// TwinCAT 3 PLC project FMS_205
// ProgramVersion: 3.1.4023.0
// libraries:
//   Tc2_Standard, * (Beckhoff Automation GmbH)
//   Tc2_System, * (Beckhoff Automation GmbH)
//   Tc3_Module, * (Beckhoff Automation GmbH)
//   VisuDialogs, * (System)
// project tree:
//   DUTs/ CaracteristicasPieza.TcDUT, E_GEMMA.TcTLEO, Pieza.TcDUT
//   / GlobalTextList.TcGTLO, PlcTask.TcTTO, Visualization Manager.TcVMO (not stored)
//   GVLs/ Constantes.TcGVL
//   POUs/Estacion/ FB_Coordinador_SFC.TcPOU, FB_Director.TcPOU, FB_Estacion.TcPOU
//   POUs/FBs/ FB_Clock.TcPOU
//   POUs/Funciones/ AjustarIndice.TcPOU
//   POUs/ MAIN.TcPOU
//   POUs/Tareas/ FB_AvanzarAlimentador_SFC.TcPOU, FB_EstacionVaciar_SFC.TcPOU, FB_EstacionRestaurar_SFC.TcPOU, FB_Medir_SFC.TcPOU, FB_EmpujarPlato_SFC.TcPOU, FB_RechazarPieza_SFC.TcPOU, FB_DescargarPieza_SFC.TcPOU, FB_SituarPale_SFC.TcPOU, FB_CargarPieza_SFC.TcPOU, FB_TransferirPale_SFC.TcPOU, FB_RetrocederPlato_SFC.TcPOU
//   VISUs/ Visualization.TcVIS
// real-time tasks:
//   TASK PlcTask: cycle T#10ms, priority 20, ADS port 350
// I/O:
//   DEVICE Device 1 (EtherCAT), AmsNetId 192.168.109.1.2.1
//     Term 1 (EK1200) [EK1200-5000 EtherCAT Power supply (2A E-Bus)]
//       Term 2 (EL1008) [EL1008 8Ch. Dig. Input 24V, 3ms]
//       Term 3 (EL1008) [EL1008 8Ch. Dig. Input 24V, 3ms]
//       Term 4 (EL2008) [EL2008 8Ch. Dig. Output 24V, 0.5A]
//       Term 5 (EL2008) [EL2008 8Ch. Dig. Output 24V, 0.5A]
//       Term 6 (EL1008) [EL1008 8Ch. Dig. Input 24V, 3ms]
//       Term 7 (EL1008) [EL1008 8Ch. Dig. Input 24V, 3ms]
//       Term 8 (EL2008) [EL2008 8Ch. Dig. Output 24V, 0.5A]
//       Term 9 (EL2008) [EL2008 8Ch. Dig. Output 24V, 0.5A]
//       Term 10 (EL5151) [EL5151 1Ch. Inc. Encoder]
//       Term 11 (EL9011) [EL9011 End Terminal]
//   DEVICE Device 3 (RT-Ethernet Protocol), AmsNetId 192.168.109.1.4.1
//   DEVICE Device 2 (NOV-DP-RAM)
// variable links:
//   FMS_205/FMS_205 Instance <-> Device 1 (EtherCAT)/Term 1 (EK1200)/Term 10 (EL5151)
//     PlcTask Inputs/MAIN.Estacion.Codificador <-> ENC Inputs/Counter value
//   FMS_205/FMS_205 Instance <-> Device 1 (EtherCAT)/Term 1 (EK1200)/Term 2 (EL1008)
//     PlcTask Inputs/MAIN.Estacion.CodigoPaleBit0 <-> Channel 7/CodigoPaleBit0
//     PlcTask Inputs/MAIN.Estacion.CodigoPaleBit1 <-> Channel 8/CodigoPaleBit1
//     PlcTask Inputs/MAIN.Estacion.EstacionConectada <-> Channel 5/EstacionConectada
//     PlcTask Inputs/MAIN.Estacion.PresenciaPale <-> Channel 6/PresenciaPale
//     PlcTask Inputs/MAIN.Estacion.PulsadorEmergencia <-> Channel 1/PulsadorEmergencia
//     PlcTask Inputs/MAIN.Estacion.PulsadorMarcha <-> Channel 3/PulsadorMarcha
//     PlcTask Inputs/MAIN.Estacion.PulsadorParada <-> Channel 4/PulsadorParada
//     PlcTask Inputs/MAIN.Estacion.SelectorManual <-> Channel 2/SelectorManual
//   FMS_205/FMS_205 Instance <-> Device 1 (EtherCAT)/Term 1 (EK1200)/Term 3 (EL1008)
//     PlcTask Inputs/MAIN.Estacion.CodigoPaleBit2 <-> Channel 1/CodigoPaleBit2
//   FMS_205/FMS_205 Instance <-> Device 1 (EtherCAT)/Term 1 (EK1200)/Term 4 (EL2008)
//     PlcTask Outputs/MAIN.Estacion.CintaActiva <-> Channel 5/CintaActiva
//     PlcTask Outputs/MAIN.Estacion.CintaInvierte <-> Channel 6/CintaInvierte
//     PlcTask Outputs/MAIN.Estacion.DesconectaEstacion <-> Channel 1/DesconectaEstacion
//     PlcTask Outputs/MAIN.Estacion.LamparaAlarma <-> Channel 2/LamparaAlarma
//     PlcTask Outputs/MAIN.Estacion.LamparaMarcha <-> Channel 3/LamparaMarcha
//     PlcTask Outputs/MAIN.Estacion.LamparaMaterial <-> Channel 4/LamparaMaterial
//     PlcTask Outputs/MAIN.Estacion.RetenedorBaja <-> Channel 7/RetenedorBaja
//     PlcTask Outputs/MAIN.Estacion.SeparadorSube <-> Channel 8/Output
//   FMS_205/FMS_205 Instance <-> Device 1 (EtherCAT)/Term 1 (EK1200)/Term 5 (EL2008)
//     PlcTask Outputs/MAIN.Estacion.AvisadorSonoro <-> Channel 1/AvisadorSonoro
//   FMS_205/FMS_205 Instance <-> Device 1 (EtherCAT)/Term 1 (EK1200)/Term 6 (EL1008)
//     PlcTask Inputs/MAIN.Estacion.CargadorAbajo <-> Channel 4/CargadorAbajo
//     PlcTask Inputs/MAIN.Estacion.CargadorArriba <-> Channel 3/CargadorArriba
//     PlcTask Inputs/MAIN.Estacion.CargadorDelante <-> Channel 2/CargadorDelante
//     PlcTask Inputs/MAIN.Estacion.CargadorDetras <-> Channel 1/CargadorDetras
//     PlcTask Inputs/MAIN.Estacion.PlatoEmpujadorDetras <-> Channel 5/PlatoEmpujadorDetras
//     PlcTask Inputs/MAIN.Estacion.RechazadorArriba <-> Channel 8/RechazadorArriba
//     PlcTask Inputs/MAIN.Estacion.RechazadorDelante <-> Channel 7/RechazadorDelante
//     PlcTask Inputs/MAIN.Estacion.RechazadorDetras <-> Channel 6/RechazadorDetras
//   FMS_205/FMS_205 Instance <-> Device 1 (EtherCAT)/Term 1 (EK1200)/Term 7 (EL1008)
//     PlcTask Inputs/MAIN.Estacion.AlimentadorDelante <-> Channel 6/AlimentadorDelante
//     PlcTask Inputs/MAIN.Estacion.DescargadorAbajo <-> Channel 5/DescargadorAbajo
//     PlcTask Inputs/MAIN.Estacion.DescargadorArriba <-> Channel 4/DescargadorArriba
//     PlcTask Inputs/MAIN.Estacion.DescargadorDelante <-> Channel 3/DescaradorDelante
//     PlcTask Inputs/MAIN.Estacion.DescargadorDetras <-> Channel 2/DescargadorDetras
//     PlcTask Inputs/MAIN.Estacion.DetectorFotoelectrico <-> Channel 8/DetectorFotoelectrico
//     PlcTask Inputs/MAIN.Estacion.DetectorInductivo <-> Channel 7/DetectorInductivo
//     PlcTask Inputs/MAIN.Estacion.RechazadorVacio <-> Channel 1/RechazadorVacio
//   FMS_205/FMS_205 Instance <-> Device 1 (EtherCAT)/Term 1 (EK1200)/Term 8 (EL2008)
//     PlcTask Outputs/MAIN.Estacion.CargadorAvanza <-> Channel 1/CargadorAvanza
//     PlcTask Outputs/MAIN.Estacion.CargadorBaja <-> Channel 2/CargadorBaja
//     PlcTask Outputs/MAIN.Estacion.CargadorCierra <-> Channel 3/CargadorCierra
//     PlcTask Outputs/MAIN.Estacion.PlatoEmpujadorAvanza <-> Channel 4/PlatoEmpujadorAvanza
//     PlcTask Outputs/MAIN.Estacion.PlatoRetenedorAtras <-> Channel 5/PlatoRetenedorAtras
//     PlcTask Outputs/MAIN.Estacion.RechazadorAvanza <-> Channel 6/RechazadorAvanza
//     PlcTask Outputs/MAIN.Estacion.RechazadorBaja <-> Channel 8/RechazadorBaja
//     PlcTask Outputs/MAIN.Estacion.RechazadorRetrocede <-> Channel 7/RechazadorRetrocede
//   FMS_205/FMS_205 Instance <-> Device 1 (EtherCAT)/Term 1 (EK1200)/Term 9 (EL2008)
//     PlcTask Outputs/MAIN.Estacion.AlimentadorAvanza <-> Channel 5/AlimentadorAvanza
//     PlcTask Outputs/MAIN.Estacion.DescargadorAvanza <-> Channel 2/DescargadorAvanza
//     PlcTask Outputs/MAIN.Estacion.DescargadorBaja <-> Channel 3/DescargadorBaja
//     PlcTask Outputs/MAIN.Estacion.DescargadorCierra <-> Channel 4/DescargadorCierra
//     PlcTask Outputs/MAIN.Estacion.MedidorBaja <-> Channel 6/MedidorBaja
//     PlcTask Outputs/MAIN.Estacion.RechazadorSucciona <-> Channel 1/RechazadorSucciona

CONFIGURATION FMS_205
    RESOURCE PLC ON TwinCAT3
        TASK PlcTask(INTERVAL := T#10ms, PRIORITY := 20);
        PROGRAM MAIN WITH PlcTask : MAIN;
    END_RESOURCE
END_CONFIGURATION

// ---- DUTs/CaracteristicasPieza.TcDUT
TYPE CaracteristicasPieza:
STRUCT
    Claro     : BOOL := FALSE;
    Metalico  : BOOL := FALSE;
	Alta : BOOL := FALSE;				//1290 Alta , 1370 baja. Reves: >1685 No hay >2000
END_STRUCT
END_TYPE

// ---- DUTs/E_GEMMA.TcTLEO
{attribute 'qualified_only'}
{attribute 'strict'}
TYPE E_GEMMA :
(
    // Modos de la Guia de Estudio de los Modos de Marcha y Parada
    // Modes du Guide d'Etude des Modes de Marche et d'Arrêt
    // Modes of Study Guide of the Modes of Operating and Stopping

    // Procedimientos de parada [Les procédures d'arrets - Stop procedure
    A1, //  0: Parada en el estado inicial 
        //  0: Arrêt dans etat initial
        //  0: Stopped in the initial state
    A2, //  1: Parada solicitada a final de ciclo 
        //  1: Arret demandé en fin de cycle
        //  1: Requested end cycle stop
    A3, //  2: Parada solicitada en un estado determinado 
        //  2: Arret demande dans etat determine
        //  2: Requested particular state stop
    A4, //  3: Parada obtenida 
        //  3: Arret obtenu 
        //  3: Obteined stop
    A5, //  4: Preparacion para la recuperacion del fallo 
        //  4: Preparation pour remise en route apres defaillance
        //  4: Preparation for the recovery of the failure
    A6, //  5: Situando la PO en el estado inicial 
        //  5: Mise PO dans état initial 
        //  5: Set the PO in initial state
    A7, //  6: Situando la PO en un estado determinado 
        //  6: Mise PO dans état déterminé 
        //  6: Set the PO in a certain state

    // Procedimientos de funcionamiento 
    // Les procédures de fonctionnement 
    // Operating procedures
    F1, //  7: Produccion normal 
        //  7: Production normale 
        //  7: Normal operation
    F2, //  8: Secuencia de preparacion 
        //  8: Marche de preparation 
        //  8: Preparation sequence
    F3, //  9: Secuencia de finalizacion 
        //  9: Marche de cloture
        //  9: Ending sequence
    F4, // 10: Verificacion en desorden 
        // 10: Marche de verification dans le desordre 
        // 10: Verification with no order
    F5, // 11: Verificacion en orden 
        // 11: Marche de verification dans l'ordre 
        // 11: Verification whit order
    F6, // 12: Secuencia de prueba 
        // 12: Marche de test 
        // 12:Test sequence

    // Procedimientos de fallo 
    // es procédures en défaillances
    // Failure procedures
    D1, // 13: Parada de emergencia 
        // 13: Arret d'urgence 
        // 13: Emergency stop
    D2, // 14: Diagnostico y/o tratamiento de los fallos 
        // 14: Diagnostic et/ou traitement de la défaillance 
        // 14: Diagnosis and/or treatment of failures
    D3  // 15: Produccion a pesar de los fallos 
        // 15: Production tout de même 
        // 15: Production despite the failures
);
END_TYPE

// ---- DUTs/Pieza.TcDUT
TYPE Pieza:
STRUCT
    TipoPieza : CaracteristicasPieza;		
	BienColocada    : BOOL := FALSE;
	EsBuena : BOOL := FALSE;
END_STRUCT
END_TYPE

// ---- GVLs/Constantes.TcGVL
VAR_GLOBAL CONSTANT
	TAMANO_LISTA_PIEZAS : UINT := 8;
	TAMANO_LISTA_CONDICIONES : UINT := 6;
END_VAR

// ---- POUs/MAIN.TcPOU
PROGRAM MAIN
//Ingenieria Electronica Robotica y Mecatronica (GIERM)
//Autmatizacion Industrial
//FMS205 
//GEMMA
//Grupo 03
//Paula Chova Garcia
//Jose Luis Perez Martin
//Tobias Garibaldi Thwaites Rayner


VAR
    Estacion: FB_Estacion;
END_VAR

Estacion();

END_PROGRAM

// ---- POUs/Estacion/FB_Estacion.TcPOU
FUNCTION_BLOCK FB_Estacion
// FMS-203 - Estructurado
VAR CONSTANT
	
END_VAR
VAR_INPUT
    // Parametros de control de la estacion
    CicloACiclo: BOOL := 0;
	PausaEstado: BOOL;
    ReiniciaEstado: BOOL;   
	FinCiclo: BOOL := FALSE;
	PiezaAPieza: BOOL := FALSE;
	FinPieza: BOOL:= FALSE;
	Fallo: BOOL := FALSE;
	FaltaMaterial : BOOL := FALSE;

    // Parametros de control de la tarea
    UnidadesSolicitadas: UINT := 1;
    
	//Variables auxiliares
	NCiclos : INT := 0;
	
    // Parametros de tiempo
    TpoPinza: TIME := T#1S;
	TpoRechazador: TIME := T#1S;
	TpoEmpujadorAvanza: TIME := T#1S;
    TpoPaleEntrada: TIME := T#1S;
	TpoPaleSalida : TIME := T#1S;
	TpoCintaRetenedor : TIME := T#1S;
	TpoPaleTransferencia : TIME := T#1S;
	TpoAlimentador: TIME := T#1300MS;
    TpoMedidor: TIME := T#1S;
	TpoPreparacion: TIME := T#1S;
	TpoFinalizacion : TIME := T#2S;
    
END_VAR

VAR_OUTPUT
	  // Parametros de; estado de la estacion
    CondicionInicial: BOOL;
    CondicionMarcha: BOOL;
	PrepararProduccion: BOOL := FALSE;
	FinalizarProduccion: BOOL := FALSE;
    CodigoPale: BYTE;  
    
    // Parametros de control de la tarea 
    UnidadesPendientes: UINT := 0;
    UnidadesRealizadas: UINT :=0;
	
	 // Entradas comunes
    PulsadorEmergencia AT %I*: BOOL;
    SelectorManual AT %I*: BOOL;
    PulsadorMarcha AT %I*: BOOL;
    PulsadorParada AT %I*: BOOL := TRUE; // Contacto normalmente cerrado
    EstacionConectada AT %I*: BOOL := TRUE;
    PresenciaPale AT %I*: BOOL;
    CodigoPaleBit0 AT %I*: BOOL;
    CodigoPaleBit1 AT %I*: BOOL;
    CodigoPaleBit2 AT %I*: BOOL;

    // Entradas espeficicas
    CargadorDetras AT %I*: BOOL;
	CargadorDelante AT %I*: BOOL;
	CargadorArriba AT %I*: BOOL;
	CargadorAbajo AT %I*: BOOL;
	PlatoEmpujadorDetras AT %I*: BOOL;
	RechazadorDetras AT %I*: BOOL;
	RechazadorDelante AT %I*: BOOL;
	RechazadorArriba AT %I*: BOOL;
	
	RechazadorVacio AT %I*: BOOL;
	DescargadorDetras AT %I*: BOOL;
	DescargadorDelante AT %I*: BOOL;
	DescargadorArriba AT %I*: BOOL;
	DescargadorAbajo AT %I*: BOOL;
	AlimentadorDelante AT %I*: BOOL := FALSE;
	DetectorInductivo AT %I*: BOOL;
	DetectorFotoelectrico AT %I*: BOOL;
	Codificador AT %I*: UINT;
END_VAR

VAR
	ModoAnterior: E_GEMMA; 
	
	 // Bloques funcionales
	CLK: FB_Clock;
	
	Director: FB_Director;
    Coordinador: FB_Coordinador_SFC;
	
	Restaurar: FB_EstacionRestaurar_SFC;
    Vaciar: FB_EstacionVaciar_SFC;
	AvanzarAlimentador: FB_AvanzarAlimentador_SFC;
    SituarPale: FB_SituarPale_SFC;
    CargarPieza: FB_CargarPieza_SFC;
	EmpujarPlato: FB_EmpujarPlato_SFC;
	RetrocederPlato : FB_RetrocederPlato_SFC;
    DescargarPieza: FB_DescargarPieza_SFC;
    RechazarPieza: FB_RechazarPieza_SFC;
    TransferirPale: FB_TransferirPale_SFC;
	Medir: FB_Medir_SFC;
	
	// Arrays
	ListadePiezas: ARRAY[1..TAMANO_LISTA_PIEZAS] OF Pieza; // Array de tamaño 8 piezas 
	ListaPiezasSolicitadas: ARRAY[1..TAMANO_LISTA_CONDICIONES] OF UINT
 	:= [TAMANO_LISTA_CONDICIONES(0)]; 
	
    // Salidas comunes
    DesconectaEstacion AT %Q*: BOOL;
    LamparaAlarma AT %Q*: BOOL;
    LamparaMarcha AT %Q*: BOOL;
	LamparaMaterial AT %Q*: BOOL;
    CintaActiva AT %Q*: BOOL;
    CintaInvierte AT %Q*: BOOL;
    RetenedorBaja AT %Q*: BOOL;
	
	AvisadorSonoro AT %Q*: BOOL;

    // Salidas especificas
    CargadorAvanza AT %Q*: BOOL;
	CargadorBaja AT %Q*: BOOL; 	
	CargadorCierra AT %Q*: BOOL;
	PlatoEmpujadorAvanza AT %Q*: BOOL;
	PlatoRetenedorAtras AT %Q*: BOOL;
	RechazadorAvanza AT %Q*: BOOL;
	RechazadorRetrocede AT %Q*: BOOL;
	RechazadorBaja AT %Q*: BOOL;
	
	RechazadorSucciona AT %Q*: BOOL;
	DescargadorAvanza AT %Q*: BOOL;
	DescargadorBaja AT %Q*: BOOL;
	DescargadorCierra AT %Q*: BOOL;
	AlimentadorAvanza AT %Q*: BOOL;
	MedidorBaja AT %Q*: BOOL;
	SeparadorSube AT %Q*: BOOL;	
	
	PlatoEmpujado: BOOL;
	PiezaRechazada: BOOL;
END_VAR

Director(
	CondicionInicial := CondicionInicial,
    CondicionMarcha := CondicionMarcha,
	Emergencia := PulsadorEmergencia,
    FaltaPreparacion := (UnidadesRealizadas = 0) AND Director.Modo = E_GEMMA.A1,
    FinTarea := (UnidadesPendientes = 0),
    FinCiclo := Coordinador.Done,
	FinPieza := FinPieza,
    Manual := SelectorManual,
    Marcha := PulsadorMarcha,
    ParaCiclo := NOT PulsadorParada,
    Preparada := Vaciar.Done,
    Reinicia := ReiniciaEstado,
	PrepararProduccion := PrepararProduccion,
    FinalizarProduccion := FinalizarProduccion,
	Fallo := Fallo
);

// MODO AUTOMATICO
IF (Director.Modo <> E_GEMMA.F4) THEN
    // Bloques funcionales
    Coordinador(
        SFCPause := NOT ReiniciaEstado AND PausaEstado, 
        // OR Director.Modo := E_GEMMA.F3 
        SFCReset := ReiniciaEstado,
        Ack := TRUE,
        Execute :=  (Director.Modo = E_GEMMA.F1),
        Resume := PulsadorMarcha,
        StepByStep := CicloaCiclo,
		FinCiclo := FinCiclo,
		FinPieza => FinPieza,
		PiezaAPieza := PiezaAPieza,
        PaleSituado := SituarPale.Done,
		AlimentadorAvanzado := AvanzarAlimentador.Done,
        PiezaCargada := CargarPieza.Done,
        PlatoEmpujado := EmpujarPlato.Done,
		PlatoRetrocedido := RetrocederPlato.Done,
        PiezaDescargada := DescargarPieza.Done,
        PiezaRechazada := RechazarPieza.Done,
		PiezaMedida := Medir.Done,
        PaleTransferido := TransferirPale.Done,
        CondicionInicial := CondicionInicial,
        UnidadesSolicitadas => UnidadesSolicitadas,
		UnidadesRealizadas => UnidadesRealizadas,
		UnidadesPendientes => UnidadesPendientes,
		ListadePiezas := ListadePiezas,
		ListaPiezasSolicitadas := ListaPiezasSolicitadas,
		Fallo => Fallo,
		FaltaMaterial := FaltaMaterial
        );
        
    SituarPale(
        SFCPause := NOT ReiniciaEstado AND PausaEstado,
        SFCReset := ReiniciaEstado,
        Ack := NOT Coordinador.SituaPale,
        Execute := Coordinador.SituaPale,
        TpoPaleEntrada := TpoPaleEntrada,
        PresenciaPale := PresenciaPale,
        CodigoPaleBit0 := CodigoPaleBit0,
        CodigoPaleBit1 := CodigoPaleBit1,
        CodigoPaleBit2 := CodigoPaleBit2
        );
        
	 AvanzarAlimentador(
        SFCPause := NOT ReiniciaEstado AND PausaEstado,
        SFCReset := ReiniciaEstado,
        Ack := NOT Coordinador.AvanzaAlimentador,
        Execute := Coordinador.AvanzaAlimentador,
		TpoAlimentador :=  TpoAlimentador,
        AlimentadorDelante := AlimentadorDelante,
		PulsadorMarcha := PulsadorMarcha,
		Fallo => Fallo,
		FaltaMaterial := FaltaMaterial
        );	
	

    CargarPieza(
        SFCPause := NOT ReiniciaEstado AND PausaEstado,
        SFCReset := ReiniciaEstado,
        Ack := NOT Coordinador.CargaPieza,
        Execute := Coordinador.CargaPieza,
		TpoPinza :=  TpoPinza,
        CargadorDetras := CargadorDetras,
		CargadorDelante := CargadorDelante,
		CargadorArriba := CargadorArriba,
		CargadorAbajo := CargadorAbajo
        );
        
     EmpujarPlato(
        SFCPause := NOT ReiniciaEstado AND PausaEstado,
        SFCReset := ReiniciaEstado,
        Ack := NOT Coordinador.EmpujaPlato AND NOT Vaciar.EmpujaPlato,
        Execute := Coordinador.EmpujaPlato OR Vaciar.EmpujaPlato,
		TpoEmpujadorAvanza := TpoEmpujadorAvanza,
        );
	
	RetrocederPlato(
        SFCPause := NOT ReiniciaEstado AND PausaEstado,
        SFCReset := ReiniciaEstado,
        Ack := NOT Coordinador.RetrocederPlato,
        Execute := Coordinador.RetrocederPlato,
		TpoEmpujadorAvanza :=  TpoEmpujadorAvanza,
        PlatoEmpujadorDetras := PlatoEmpujadorDetras,
        );
		
    
    DescargarPieza(
        SFCPause := NOT ReiniciaEstado AND PausaEstado,
        SFCReset := ReiniciaEstado,
        Ack := NOT Coordinador.DescargaPieza,
        Execute := Coordinador.DescargaPieza,
        TpoPinza :=  TpoPinza,
        DescargadorDetras := DescargadorDetras,
        DescargadorDelante := DescargadorDelante,
        DescargadorArriba := DescargadorArriba,
        DescargadorAbajo := DescargadorAbajo
        );
    
    RechazarPieza(
        SFCPause := NOT ReiniciaEstado AND PausaEstado,
        SFCReset := ReiniciaEstado,
        Ack := NOT Coordinador.RechazaPieza AND NOT Vaciar.RechazaPieza,
        Execute := Coordinador.RechazaPieza OR Vaciar.RechazaPieza,
		TpoRechazador := TpoRechazador,
        RechazadorDetras := RechazadorDetras,
        RechazadorDelante := RechazadorDelante,
        RechazadorArriba := RechazadorArriba,
		RechazadorVacio := RechazadorVacio,
		PulsadorMarcha := PulsadorMarcha,
		Fallo => Fallo
        );
		
	 Medir(
        SFCPause := NOT ReiniciaEstado AND PausaEstado,
        SFCReset := ReiniciaEstado,
        Ack := NOT Coordinador.MedidorMide,
        Execute := Coordinador.MedidorMide,
		TpoMedidor := TpoMedidor,
        Codificador := Codificador,
        DetectorFotoelectrico := DetectorFotoelectrico,
        DetectorInductivo := DetectorInductivo,
		NCiclos := NCiclos,
		ListadePiezas := ListadePiezas,
        );
    
    TransferirPale(
        SFCPause := NOT ReiniciaEstado AND PausaEstado,
        SFCReset := ReiniciaEstado,
        Ack := NOT Coordinador.TransfierePale,
        Execute := Coordinador.TransfierePale,
        TpoCintaRetenedor := TpoCintaRetenedor,
        TpoPaleSalida := TpoPaleSalida,
        TpoPaleTransferencia := TpoPaleTransferencia,
        PresenciaPale := PresenciaPale
        );
    Restaurar(
        SFCPause := NOT ReiniciaEstado AND PausaEstado,
        SFCReset := ReiniciaEstado,
        Ack := TRUE,
        Execute := (Director.Modo = E_GEMMA.A6),
        CargadorDetras := CargadorDetras,
        PlatoEmpujadorDetras := PlatoEmpujadorDetras,
        DescargadorDetras := DescargadorDetras,
		RechazadorDetras := RechazadorDetras
        );
	Vaciar(
        SFCPause := NOT ReiniciaEstado AND PausaEstado,
        SFCReset := ReiniciaEstado,
        Ack := (Director.Modo <> E_GEMMA.F2) AND (Director.Modo <> E_GEMMA.F3),
        Execute := (Director.Modo = E_GEMMA.F2) OR (Director.Modo = E_GEMMA.F3),
		TpoPreparacion := TpoPreparacion,
        TpoMedidor := TpoMedidor,
		PlatoEmpujado := EmpujarPlato.Done,
		PiezaRechazada := RechazarPieza.Done,
		PulsadorMarcha := PulsadorMarcha,
		Codificador := Codificador
        );
		
    // Acciones
   AvisadorSonoro := ((Director.Modo = E_GEMMA.F2) AND CLK.Q) 
        OR (Director.Modo = E_GEMMA.F3)
		OR (Director.Modo = E_GEMMA.D1)
		OR (Director.Modo = E_GEMMA.D2);   
    LamparaAlarma := (Director.Modo = E_GEMMA.D1) 
        OR ((Director.Modo = E_GEMMA.A6) AND CLK.Q)
		OR (Director.Modo = E_GEMMA.D2);
    LamparaMarcha := (Director.Produccion AND NOT Coordinador.Done)
        OR ((Director.Modo = E_GEMMA.A1) AND CLK.Q);
    

    CintaActiva := NOT PausaEstado 
        AND (SituarPale.CintaActiva OR TransferirPale.CintaActiva);
    RetenedorBaja := TransferirPale.RetenedorBaja;
	SeparadorSube := TransferirPale.SeparadorSube;
	AlimentadorAvanza := AvanzarAlimentador.AlimentadorAvanza;
    CargadorAvanza := CargarPieza.CargadorAvanza; 
    CargadorBaja := CargarPieza.CargadorBaja;    
	CargadorCierra := CargarPieza.CargadorCierra;
	PlatoEmpujadorAvanza := EmpujarPlato.PlatoEmpujadorAvanza;
	PlatoRetenedorAtras := EmpujarPlato.PlatoRetenedorAtras;
	DescargadorAvanza := DescargarPieza.DescargadorAvanza; 
    DescargadorBaja := DescargarPieza.DescargadorBaja;    
	DescargadorCierra := DescargarPieza.DescargadorCierra;
    RechazadorAvanza := RechazarPieza.RechazadorAvanza;
	RechazadorSucciona := RechazarPieza.RechazadorSucciona;
    RechazadorRetrocede := RechazarPieza.RechazadorRetrocede
	OR Restaurar.RechazadorRetrocede;
    RechazadorBaja := RechazarPieza.RechazadorBaja;
	AlimentadorAvanza := AvanzarAlimentador.AlimentadorAvanza;
	MedidorBaja := Medir.MedidorBaja OR Vaciar.MedidorBaja;
	
   
END_IF

// Parametros de salida
CondicionInicial := EstacionConectada 
    AND CargadorDetras 
    AND PlatoEmpujadorDetras
    AND DescargadorDetras
    AND RechazadorDetras;

CondicionMarcha := (UnidadesSolicitadas > 0);
NCiclos := Coordinador.NCiclos;


IF (Director.Modo <> E_GEMMA.F4) THEN
    CodigoPale := SituarPale.CodigoPale;
ELSE 
    CodigoPale.0 := CodigoPaleBit0;
    CodigoPale.1 := CodigoPaleBit1;
    CodigoPale.2 := CodigoPaleBit2;
END_IF

// ACTULIZACION DE IMAGENES
ModoAnterior := Director.Modo;

END_FUNCTION_BLOCK

// ---- POUs/FBs/FB_Clock.TcPOU
FUNCTION_BLOCK FB_Clock
(*
Square wave oscillator

Copyright (c) 2009-2017 victortorreslopez

GNU General Public License

Version history
2.1, 2017/03/15, VTL: style review (PLCopen Coding Guidelines)
2.0, 2014/12/29, VTL: complete review
1.0, 2009/11/06, VTL: first release
0.0, 2009/11/06, VTL: alfa release
*)
VAR_INPUT
  EN: BOOL := TRUE;	(* ENabled *)
  PT: TIME := T#500ms; (* Semicycle time *)
END_VAR
VAR_OUTPUT
  ET: TIME; (* Elapsed time *)
  Q: BOOL; (* Square wave *)
END_VAR
VAR
  Timer: TON; (* Auto-pilot timer *)
END_VAR

(* OUTPUT FUNCTION *)
IF Timer.Q THEN
  Q := NOT Q;
END_IF

(* FUNCTION BLOCKS *)
Timer(IN := EN AND NOT Timer.Q, PT := PT, ET => ET);

END_FUNCTION_BLOCK

// ---- POUs/Estacion/FB_Director.TcPOU
FUNCTION_BLOCK FB_Director
// FMS-203 - GEMMA

VAR_INPUT
    CondicionInicial: BOOL;
    CondicionMarcha: BOOL; 
    Emergencia: BOOL;
    FinTarea: BOOL;
    FinCiclo: BOOL;
	FinPieza: BOOL;
    Manual: BOOL;
    Marcha: BOOL;
    ParaCiclo: BOOL;
    Preparada: BOOL;
    Reinicia: BOOL;
	Fallo: BOOL;
	PrepararProduccion: BOOL;
    FinalizarProduccion: BOOL;
    FaltaPreparacion: BOOL;
END_VAR
VAR_OUTPUT
    Modo: E_GEMMA := E_GEMMA.A6;

    Defecto: BOOL; // Procedimientos de defecto
    Funcionamiento: BOOL; // Procedimientos de funcionamiento
    Parada: BOOL; // Procedimientos de parada
    Produccion: BOOL; // Procedimientos que proporcionan valor añadido
END_VAR

// FUNCION DE ESTADO
IF Emergencia THEN
    Modo := E_GEMMA.D1;
ELSIF Reinicia THEN
    Modo := E_GEMMA.A6;
ELSE
    CASE Modo OF
        // Procedimientos de parada
        E_GEMMA.A1: // Parada en el estado inicial
            IF NOT CondicionInicial THEN
                Modo := E_GEMMA.A6;
            ELSIF CondicionInicial AND CondicionMarcha AND Marcha THEN
                IF FaltaPreparacion THEN 
                    Modo := E_GEMMA.F2;
                ELSE   
                    Modo := E_GEMMA.F1;
                END_IF
            ELSIF Manual THEN
                Modo := E_GEMMA.F4;
            END_IF
        E_GEMMA.A2: // Parada solicitada a final de ciclo
           IF Marcha THEN 
               Modo := E_GEMMA.F1;
		   END_IF
        E_GEMMA.A3: // Parada solicitada en un estado determinado 
       		IF Marcha THEN 
               Modo := E_GEMMA.F1;
		   END_IF   
        E_GEMMA.A4: // Parada obtenida 
            ;
        E_GEMMA.A5: // Preparando de reanudacion tras el fallo 
            ;
        E_GEMMA.A6: // Situando el sistema en el estado inicial 
            IF CondicionInicial THEN
                Modo := E_GEMMA.A1;
            ELSIF Manual THEN
                Modo := E_GEMMA.F4;
            END_IF

        // Procedimientos de funcionamiento 
        E_GEMMA.F1: // Produccion normal 
            IF FinTarea THEN
               Modo := E_GEMMA.A6;
            ELSIF FinCiclo THEN
				Modo := E_GEMMA.F3;
			ELSIF FinPieza THEN
				Modo := E_GEMMA.A2;
			ELSIF ParaCiclo THEN
               Modo := E_GEMMA.A3;
			ELSIF Fallo THEN
				Modo := E_GEMMA.D2;
			END_IF
			
        E_GEMMA.F2: // Secuencia de preparacion 
            IF Preparada AND NOT Manual THEN
                Modo := E_GEMMA.F1;
            ELSIF Preparada AND Manual THEN
                Modo := E_GEMMA.F4;
			END_IF
        E_GEMMA.F3: // Secuencia de finalizacion 
           IF Preparada AND NOT Manual THEN
                Modo := E_GEMMA.A6;
            ELSIF Preparada AND Manual THEN
                Modo := E_GEMMA.F4;
			END_IF
        E_GEMMA.F4: // Verificacion sin orden 
            IF NOT Manual THEN
                Modo := E_GEMMA.A6;
            ELSIF (CondicionInicial) AND PrepararProduccion THEN
                Modo := E_GEMMA.F2;
            ELSIF (CondicionInicial) AND FinalizarProduccion THEN
                Modo := E_GEMMA.F3;
            END_IF
        E_GEMMA.F5: // Verificacion en orden 
            ;

        // Procedimientos de defecto 
        E_GEMMA.D1: // Parada de emergencia 
            IF NOT Emergencia THEN
                Modo := E_GEMMA.A6;
            END_IF
        E_GEMMA.D2: // Diagnostico/tratamiento de los fallos 
        IF Marcha THEN
			Modo := E_GEMMA.F1;
		END_IF    
			
    END_CASE
END_IF

// PARAMETROS DE SALIDA 
Defecto := (Modo >= E_GEMMA.D1) AND (Modo <= E_GEMMA.D3);
Funcionamiento:= (Modo >= E_GEMMA.F1);
Parada := (Modo >= E_GEMMA.A1);
Produccion := (Modo = E_GEMMA.A2) 
    OR (Modo = E_GEMMA.A3) 
    OR (Modo = E_GEMMA.F1) 
    OR (Modo = E_GEMMA.F2) 
    OR (Modo = E_GEMMA.F3) 
    OR (Modo = E_GEMMA.F5)
    OR (Modo = E_GEMMA.F6) 
    OR (Modo = E_GEMMA.D3);

END_FUNCTION_BLOCK

// ---- POUs/Estacion/FB_Coordinador_SFC.TcPOU
FUNCTION_BLOCK FB_Coordinador_SFC

VAR CONSTANT
LISTA_CONDICIONES: ARRAY[1..TAMANO_LISTA_CONDICIONES] OF CaracteristicasPieza:=[(Claro:=FALSE, Metalico:=FALSE, Alta:=TRUE), //Negra alta
					(Claro:=TRUE,Metalico:=FALSE,Alta:=TRUE), //Blanca alta					
					(Claro:=TRUE, Metalico:=TRUE, Alta:=TRUE), //Metal alta
					(Claro:=FALSE, Metalico:=FALSE, Alta:=FALSE), //Negra baja
					(Claro:=TRUE, Metalico:=FALSE, Alta:=FALSE), //Blanca baja					
					(Claro:=TRUE, Metalico:=TRUE, Alta:=FALSE)]; //Metal baja
END_VAR

VAR_IN_OUT
	ListadePiezas: ARRAY[1..TAMANO_LISTA_PIEZAS] OF Pieza; // Array de tamaño 8 piezas 
	ListaPiezasSolicitadas: ARRAY[1..TAMANO_LISTA_CONDICIONES] OF UINT; // Array de 6 condiciones (blanca, negra y metálica, de momento)
	FaltaMaterial: BOOL;
END_VAR

VAR_INPUT
	  // SFC-Flags
    SFCPause: BOOL;
    SFCReset: BOOL;
    
    // Indicadores de sincronizacion
    Ack: BOOL := TRUE;
    Execute: BOOL;
    
    // Indicadores de control
    Resume: BOOL;
    StepByStep: BOOL;
	FinCiclo: BOOL;
    PiezaAPieza: BOOL;
    // Parametros de sincronizacion
    PaleSituado: BOOL;
	AlimentadorAvanzado: BOOL;
    PiezaCargada: BOOL;
	PlatoEmpujado: BOOL;
	PiezaMedida: BOOL;
    PiezaDescargada: BOOL;
    PiezaRechazada: BOOL;
    PaleTransferido: BOOL;
	PlatoRetrocedido: BOOL;
    
    // Parametros
    CondicionInicial: BOOL;

	//Variables auxiliares
	NCiclos: INT;
	AuxNciclosDesechar: INT := 1;
	AuxNciclosDescargar: INT := 1;
	ListoParaRechazar: BOOL := FALSE;
	ListoParaDescargar: BOOL := FALSE;
	ListoParaMedir: BOOL := FALSE;
	AUX_Suma_Solicitadas: UINT;
	
END_VAR
VAR_OUTPUT
	 // Indicadores de sincronizacion
    Done: BOOL;
    Ready: BOOL;
	Fallo: BOOL;
	FinPieza: BOOL;

    // Parametros de sincronizacion
    SituaPale: BOOL;
	AvanzaAlimentador: BOOL;
	EmpujaPlato: BOOL;
	MedidorMide: BOOL;
    CargaPieza: BOOL;
    DescargaPieza: BOOL;
    RechazaPieza: BOOL;
    TransfierePale: BOOL;
	RetrocederPlato: BOOL;
    
    // Salidas
    LamparaAlarma: BOOL;
    LamparaMarcha: BOOL;
	
	//Variables
	UnidadesSolicitadas: UINT := 1;
	UnidadesPendientes: UINT;
    UnidadesRealizadas: UINT; 
	
END_VAR
VAR

END_VAR

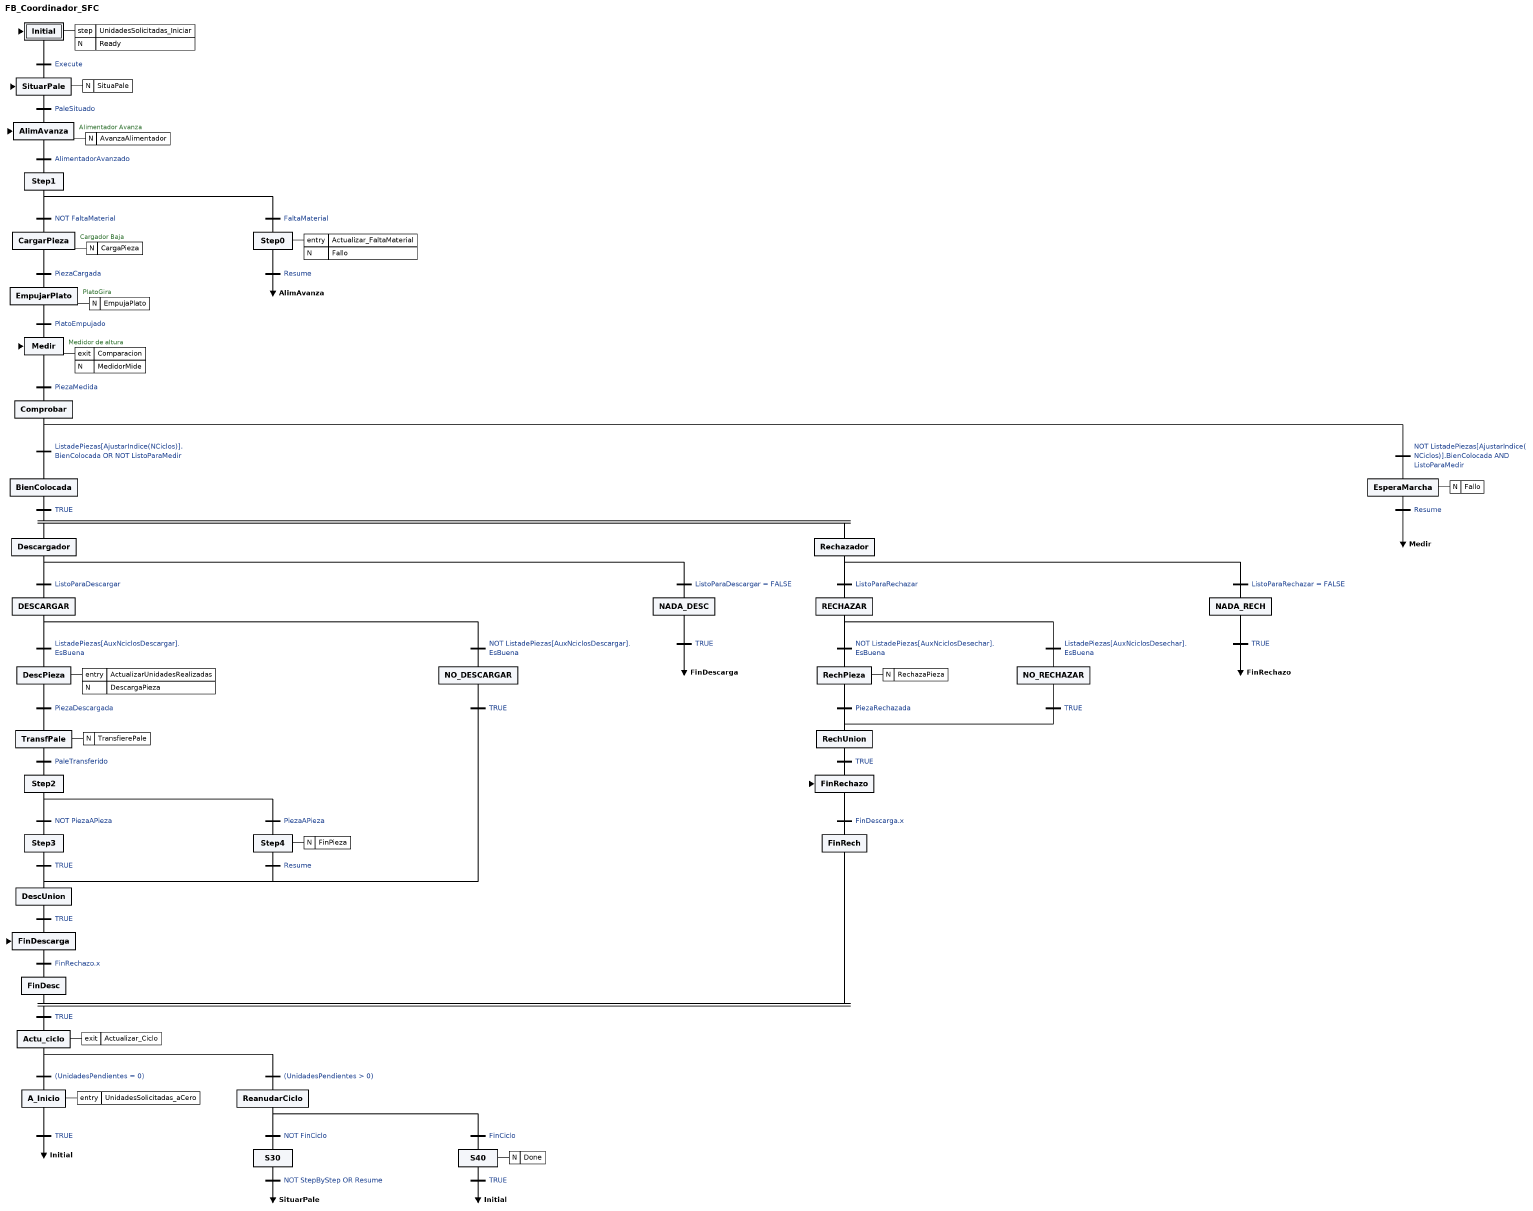
INITIAL_STEP Initial:
    UnidadesSolicitadas_Iniciar(N);  // step action
    Ready(N);
END_STEP
TRANSITION FROM Initial TO SituarPale
    := Execute;
END_TRANSITION
STEP SituarPale:
    SituaPale(N);
END_STEP
TRANSITION FROM SituarPale TO AlimAvanza
    := PaleSituado;
END_TRANSITION
// Alimentador Avanza
STEP AlimAvanza:
    AvanzaAlimentador(N);
END_STEP
TRANSITION FROM AlimAvanza TO Step1
    := AlimentadorAvanzado;
END_TRANSITION
STEP Step1:
END_STEP
TRANSITION FROM Step1 TO CargarPieza
    := NOT FaltaMaterial;
END_TRANSITION
TRANSITION FROM Step1 TO Step0
    := FaltaMaterial;
END_TRANSITION
STEP Step0:
    Actualizar_FaltaMaterial(P1);  // entry action
    Fallo(N);
END_STEP
TRANSITION FROM Step0 TO AlimAvanza
    := Resume;
END_TRANSITION
// Cargador Baja
STEP CargarPieza:
    CargaPieza(N);
END_STEP
TRANSITION FROM CargarPieza TO EmpujarPlato
    := PiezaCargada;
END_TRANSITION
// PlatoGira
STEP EmpujarPlato:
    EmpujaPlato(N);
END_STEP
TRANSITION FROM EmpujarPlato TO Medir
    := PlatoEmpujado;
END_TRANSITION
// Medidor de altura
STEP Medir:
    Comparacion(P0);  // exit action
    MedidorMide(N);
END_STEP
TRANSITION FROM Medir TO Comprobar
    := PiezaMedida;
END_TRANSITION
STEP Comprobar:
END_STEP
TRANSITION FROM Comprobar TO BienColocada
    := ListadePiezas[AjustarIndice(NCiclos)].BienColocada OR NOT ListoParaMedir;
END_TRANSITION
STEP BienColocada:
END_STEP
TRANSITION FROM BienColocada TO (Descargador, Rechazador)
    := TRUE;
END_TRANSITION
TRANSITION FROM Comprobar TO EsperaMarcha
    := NOT ListadePiezas[AjustarIndice(NCiclos)].BienColocada AND ListoParaMedir;
END_TRANSITION
STEP EsperaMarcha:
    Fallo(N);
END_STEP
TRANSITION FROM EsperaMarcha TO Medir
    := Resume;
END_TRANSITION
STEP Descargador:
END_STEP
TRANSITION FROM Descargador TO DESCARGAR
    := ListoParaDescargar;
END_TRANSITION
STEP DESCARGAR:
END_STEP
TRANSITION FROM Descargador TO NADA_DESC
    := ListoParaDescargar = FALSE;
END_TRANSITION
STEP NADA_DESC:
END_STEP
TRANSITION FROM NADA_DESC TO FinDescarga
    := TRUE;
END_TRANSITION
TRANSITION FROM DESCARGAR TO DescPieza
    := ListadePiezas[AuxNciclosDescargar].EsBuena;
END_TRANSITION
STEP DescPieza:
    ActualizarUnidadesRealizadas(P1);  // entry action
    DescargaPieza(N);
END_STEP
TRANSITION FROM DescPieza TO TransfPale
    := PiezaDescargada;
END_TRANSITION
STEP TransfPale:
    TransfierePale(N);
END_STEP
TRANSITION FROM TransfPale TO Step2
    := PaleTransferido;
END_TRANSITION
STEP Step2:
END_STEP
TRANSITION FROM Step2 TO Step3
    := NOT PiezaAPieza;
END_TRANSITION
STEP Step3:
END_STEP
TRANSITION FROM Step3 TO DescUnion
    := TRUE;
END_TRANSITION
TRANSITION FROM Step2 TO Step4
    := PiezaAPieza;
END_TRANSITION
STEP Step4:
    FinPieza(N);
END_STEP
TRANSITION FROM Step4 TO DescUnion
    := Resume;
END_TRANSITION
TRANSITION FROM DESCARGAR TO NO_DESCARGAR
    := NOT ListadePiezas[AuxNciclosDescargar].EsBuena;
END_TRANSITION
STEP NO_DESCARGAR:
END_STEP
TRANSITION FROM NO_DESCARGAR TO DescUnion
    := TRUE;
END_TRANSITION
STEP DescUnion:
END_STEP
TRANSITION FROM DescUnion TO FinDescarga
    := TRUE;
END_TRANSITION
STEP FinDescarga:
END_STEP
TRANSITION FROM FinDescarga TO FinDesc
    := FinRechazo.x;
END_TRANSITION
STEP FinDesc:
END_STEP
STEP Rechazador:
END_STEP
TRANSITION FROM Rechazador TO RECHAZAR
    := ListoParaRechazar;
END_TRANSITION
STEP RECHAZAR:
END_STEP
TRANSITION FROM Rechazador TO NADA_RECH
    := ListoParaRechazar = FALSE;
END_TRANSITION
STEP NADA_RECH:
END_STEP
TRANSITION FROM NADA_RECH TO FinRechazo
    := TRUE;
END_TRANSITION
TRANSITION FROM RECHAZAR TO RechPieza
    := NOT ListadePiezas[AuxNciclosDesechar].EsBuena;
END_TRANSITION
STEP RechPieza:
    RechazaPieza(N);
END_STEP
TRANSITION FROM RechPieza TO RechUnion
    := PiezaRechazada;
END_TRANSITION
TRANSITION FROM RECHAZAR TO NO_RECHAZAR
    := ListadePiezas[AuxNciclosDesechar].EsBuena;
END_TRANSITION
STEP NO_RECHAZAR:
END_STEP
TRANSITION FROM NO_RECHAZAR TO RechUnion
    := TRUE;
END_TRANSITION
STEP RechUnion:
END_STEP
TRANSITION FROM RechUnion TO FinRechazo
    := TRUE;
END_TRANSITION
STEP FinRechazo:
END_STEP
TRANSITION FROM FinRechazo TO FinRech
    := FinDescarga.x;
END_TRANSITION
STEP FinRech:
END_STEP
TRANSITION FROM (FinDesc, FinRech) TO Actu_ciclo
    := TRUE;
END_TRANSITION
STEP Actu_ciclo:
    Actualizar_Ciclo(P0);  // exit action
END_STEP
TRANSITION FROM Actu_ciclo TO A_Inicio
    := (UnidadesPendientes = 0);
END_TRANSITION
TRANSITION FROM Actu_ciclo TO ReanudarCiclo
    := (UnidadesPendientes > 0);
END_TRANSITION
STEP ReanudarCiclo:
END_STEP
TRANSITION FROM ReanudarCiclo TO S30
    := NOT FinCiclo;
END_TRANSITION
STEP S30:
END_STEP
TRANSITION FROM ReanudarCiclo TO S40
    := FinCiclo;
END_TRANSITION
STEP S40:
    Done(N);
END_STEP
TRANSITION FROM S40 TO Initial
    := TRUE;
END_TRANSITION
TRANSITION FROM S30 TO SituarPale
    := NOT StepByStep OR Resume;
END_TRANSITION
STEP A_Inicio:
    UnidadesSolicitadas_aCero(P1);  // entry action
END_STEP
TRANSITION FROM A_Inicio TO Initial
    := TRUE;
END_TRANSITION

ACTION Actualizar_Ciclo:
Nciclos := Nciclos + 1;
IF Nciclos >= 8 THEN // Si da una vuelta entera
   Nciclos := 0;
END_IF


// Tras 6 ciclos, la pieza puede ser desechada
IF Nciclos >= 5 THEN
   ListoParaRechazar := TRUE;
END_IF

// Tras 7 ciclos, la pieza puede ser descargada
IF  Nciclos >= 6 THEN
	ListoParaDescargar := TRUE;
END_IF

ListoParaMedir := TRUE;
END_ACTION

ACTION Actualizar_FaltaMaterial:
FaltaMaterial := FALSE;
END_ACTION

ACTION ActualizarUnidadesRealizadas:
UnidadesRealizadas := UnidadesRealizadas + 1;
UnidadesPendientes := UnidadesPendientes - 1;
END_ACTION

ACTION Comparacion:
//Si esta listo para desechar
IF ListoParaRechazar THEN
   AuxNciclosDesechar := AjustarIndice(Nciclos - 4);
	ListadePiezas[AuxNciclosDesechar].EsBuena := FALSE;
							
	IF ListadePiezas[AuxNciclosDesechar].BienColocada THEN // Evaluacion de las condiciones exigidas
		ListadePiezas[AuxNciclosDesechar].EsBuena := EvaluarPieza(Indice := AuxNciclosDesechar,
																  LISTA_CONDICIONES := LISTA_CONDICIONES,
																  ListadePiezas := ListadePiezas,
																  ListaPiezasSolicitadas := ListaPiezasSolicitadas
																  );
	END_IF
END_IF

//Si esta listo para descargar		
IF ListoParaDescargar THEN	
	AuxNciclosDescargar := AjustarIndice(Nciclos - 5);
END_IF
END_ACTION

METHOD EvaluarPieza : BOOL
VAR_INPUT
	Indice : INT;
	LISTA_CONDICIONES : ARRAY[1..TAMANO_LISTA_CONDICIONES] OF CaracteristicasPieza;
END_VAR

VAR_IN_OUT
	ListadePiezas : ARRAY[1..TAMANO_LISTA_PIEZAS] OF Pieza; 
	ListaPiezasSolicitadas: ARRAY[1..TAMANO_LISTA_CONDICIONES] OF UINT; 
END_VAR

VAR
	ContadorComparacion : INT := 1;
END_VAR
WHILE NOT ListadePiezas[Indice].EsBuena AND ContadorComparacion<7 DO 
	IF ListaPiezasSolicitadas[ContadorComparacion] > 0 THEN 
		IF MEMCMP (ADR(ListadePiezas[Indice].TipoPieza), 
			       ADR(LISTA_CONDICIONES[ContadorComparacion]), 
                   SIZEOF(LISTA_CONDICIONES[ContadorComparacion])) = 0 
       	THEN
			ListadePiezas[Indice].EsBuena := TRUE; 
            ListaPiezasSolicitadas[ContadorComparacion] := ListaPiezasSolicitadas[ContadorComparacion] - 1;
		END_IF
	END_IF
			ContadorComparacion := ContadorComparacion + 1;
END_WHILE

EvaluarPieza := ListadePiezas[Indice].EsBuena;
END_METHOD

ACTION UnidadesSolicitadas_aCero:
ListaPiezasSolicitadas[1] := 0;
ListaPiezasSolicitadas[2] := 0;
ListaPiezasSolicitadas[3] := 0;
ListaPiezasSolicitadas[4] := 0;
ListaPiezasSolicitadas[5] := 0;
ListaPiezasSolicitadas[6] := 0;
END_ACTION

ACTION UnidadesSolicitadas_Iniciar:
UnidadesSolicitadas := 0;
 
//Suma de todas las iezas solicitadas
FOR AUX_Suma_Solicitadas := 1 TO TAMANO_LISTA_CONDICIONES DO
    UnidadesSolicitadas := UnidadesSolicitadas + ListaPiezasSolicitadas[AUX_Suma_Solicitadas];
END_FOR;

    UnidadesPendientes := UnidadesSolicitadas;
END_ACTION

END_FUNCTION_BLOCK

// ---- POUs/Funciones/AjustarIndice.TcPOU
FUNCTION AjustarIndice : INT
VAR_INPUT
    ValorBase: INT;
END_VAR					//Cambiar por un Property?

IF ValorBase < 1 THEN
    AjustarIndice := ValorBase + 8;
ELSE
    AjustarIndice := ValorBase;
END_IF

END_FUNCTION

// ---- POUs/Tareas/FB_EstacionRestaurar_SFC.TcPOU
FUNCTION_BLOCK FB_EstacionRestaurar_SFC
VAR_INPUT
    // SFC-Flags
    SFCPause: BOOL;
    SFCReset: BOOL;
    
    // Indicadores de sincronizacion
    Ack: BOOL := TRUE;
    Execute: BOOL;
    
    // Entradas
    	CargadorDetras : BOOL;
        PlatoEmpujadorDetras : BOOL;
        DescargadorDetras : BOOL;
		RechazadorDetras : BOOL; 
END_VAR
VAR_OUTPUT
    // Indicadores de sincronizacion
    Done: BOOL;
    Ready: BOOL;
    
	//Sallidas
	RechazadorRetrocede : BOOL;
	
END_VAR
VAR
END_VAR

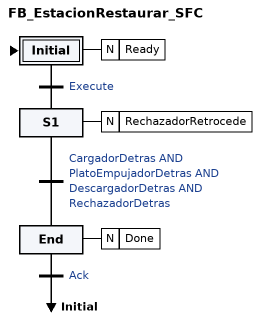
INITIAL_STEP Initial:
    Ready(N);
END_STEP
TRANSITION FROM Initial TO S1
    := Execute;
END_TRANSITION
STEP S1:
    RechazadorRetrocede(N);
END_STEP
TRANSITION FROM S1 TO End
    := CargadorDetras AND PlatoEmpujadorDetras AND DescargadorDetras AND RechazadorDetras;
END_TRANSITION
STEP End:
    Done(N);
END_STEP
TRANSITION FROM End TO Initial
    := Ack;
END_TRANSITION

END_FUNCTION_BLOCK

// ---- POUs/Tareas/FB_EstacionVaciar_SFC.TcPOU
FUNCTION_BLOCK FB_EstacionVaciar_SFC

VAR_IN_OUT
	 TpoPreparacion: TIME;
     TpoMedidor: TIME;
END_VAR

VAR_INPUT
    // SFC-Flags
    SFCPause: BOOL;
    SFCReset: BOOL;
    
    // Indicadores de sincronizacion
    Ack: BOOL:= TRUE;
    Execute: BOOL;
	
	PlatoEmpujado: BOOL;
	PiezaRechazada: BOOL;
	PulsadorMarcha: BOOL;
	PiezaMedida: BOOL;
	Codificador: UINT;
    
END_VAR
VAR_OUTPUT
    // Indicadores de sincronizacion
    Done: BOOL;
    Ready: BOOL;
	EmpujaPlato : BOOL;
	RechazaPieza : BOOL;
	MedidorBaja: BOOL;
END_VAR
VAR
	Contador: INT;
    AuxiliarContador: INT;
	ListaAlturas : ARRAY[1..TAMANO_LISTA_PIEZAS] OF UINT;
END_VAR

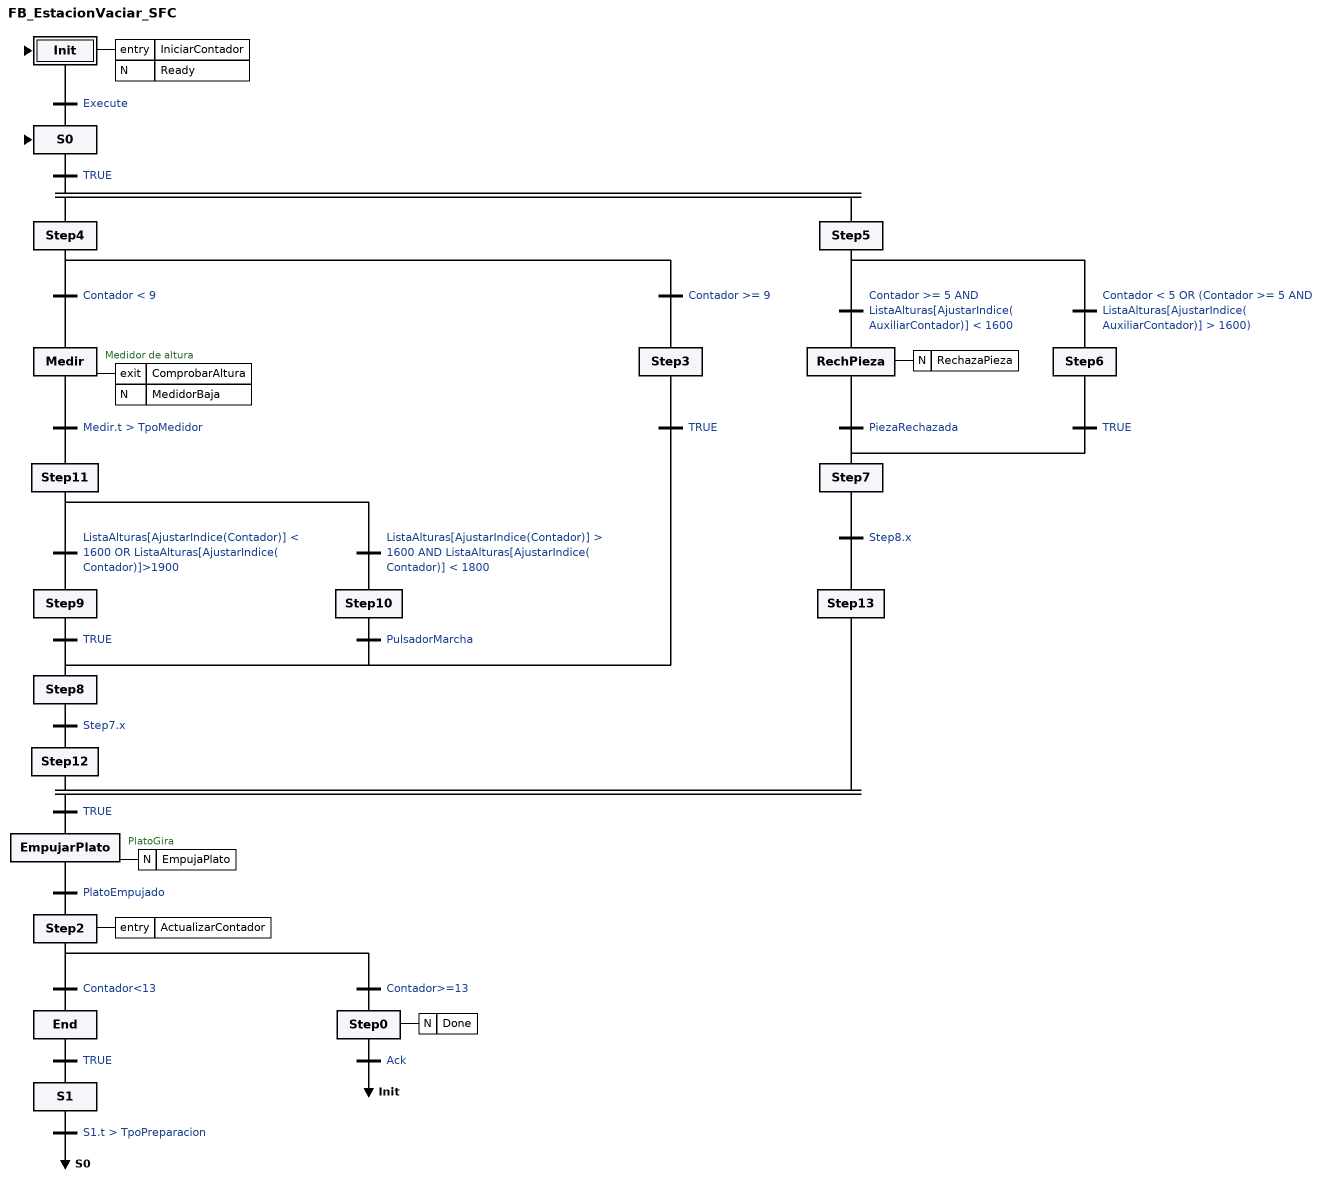
INITIAL_STEP Init:
    IniciarContador(P1);  // entry action
    Ready(N);
END_STEP
TRANSITION FROM Init TO S0
    := Execute;
END_TRANSITION
STEP S0:
END_STEP
TRANSITION FROM S0 TO (Step4, Step5)
    := TRUE;
END_TRANSITION
STEP Step4:
END_STEP
TRANSITION FROM Step4 TO Medir
    := Contador < 9;
END_TRANSITION
// Medidor de altura
STEP Medir:
    ComprobarAltura(P0);  // exit action
    MedidorBaja(N);
END_STEP
TRANSITION FROM Medir TO Step11
    := Medir.t > TpoMedidor;
END_TRANSITION
STEP Step11:
END_STEP
TRANSITION FROM Step11 TO Step9
    := ListaAlturas[AjustarIndice(Contador)] < 1600 OR ListaAlturas[AjustarIndice(Contador)]>1900;
END_TRANSITION
STEP Step9:
END_STEP
TRANSITION FROM Step9 TO Step8
    := TRUE;
END_TRANSITION
TRANSITION FROM Step11 TO Step10
    := ListaAlturas[AjustarIndice(Contador)] > 1600 AND ListaAlturas[AjustarIndice(Contador)] < 1800;
END_TRANSITION
STEP Step10:
END_STEP
TRANSITION FROM Step10 TO Step8
    := PulsadorMarcha;
END_TRANSITION
TRANSITION FROM Step4 TO Step3
    := Contador >= 9;
END_TRANSITION
STEP Step3:
END_STEP
TRANSITION FROM Step3 TO Step8
    := TRUE;
END_TRANSITION
STEP Step8:
END_STEP
TRANSITION FROM Step8 TO Step12
    := Step7.x;
END_TRANSITION
STEP Step12:
END_STEP
STEP Step5:
END_STEP
TRANSITION FROM Step5 TO RechPieza
    := Contador >= 5 AND ListaAlturas[AjustarIndice(AuxiliarContador)] < 1600;
END_TRANSITION
STEP RechPieza:
    RechazaPieza(N);
END_STEP
TRANSITION FROM RechPieza TO Step7
    := PiezaRechazada;
END_TRANSITION
TRANSITION FROM Step5 TO Step6
    := Contador < 5 OR (Contador >= 5 AND ListaAlturas[AjustarIndice(AuxiliarContador)] > 1600);
END_TRANSITION
STEP Step6:
END_STEP
TRANSITION FROM Step6 TO Step7
    := TRUE;
END_TRANSITION
STEP Step7:
END_STEP
TRANSITION FROM Step7 TO Step13
    := Step8.x;
END_TRANSITION
STEP Step13:
END_STEP
TRANSITION FROM (Step12, Step13) TO EmpujarPlato
    := TRUE;
END_TRANSITION
// PlatoGira
STEP EmpujarPlato:
    EmpujaPlato(N);
END_STEP
TRANSITION FROM EmpujarPlato TO Step2
    := PlatoEmpujado;
END_TRANSITION
STEP Step2:
    ActualizarContador(P1);  // entry action
END_STEP
TRANSITION FROM Step2 TO End
    := Contador<13;
END_TRANSITION
STEP End:
END_STEP
TRANSITION FROM End TO S1
    := TRUE;
END_TRANSITION
TRANSITION FROM Step2 TO Step0
    := Contador>=13;
END_TRANSITION
STEP Step0:
    Done(N);
END_STEP
TRANSITION FROM Step0 TO Init
    := Ack;
END_TRANSITION
STEP S1:
END_STEP
TRANSITION FROM S1 TO S0
    := S1.t > TpoPreparacion;
END_TRANSITION

ACTION ActualizarContador:
Contador := Contador + 1;
AuxiliarContador := Contador - 4;
END_ACTION

ACTION ComprobarAltura:
ListaAlturas[contador] := Codificador;
END_ACTION

ACTION IniciarContador:
Contador := 1;
END_ACTION

END_FUNCTION_BLOCK

// ---- POUs/Tareas/FB_AvanzarAlimentador_SFC.TcPOU
FUNCTION_BLOCK FB_AvanzarAlimentador_SFC

VAR_IN_OUT
	   TpoAlimentador: TIME;
	   FaltaMaterial: BOOL;
END_VAR

VAR_INPUT
    // SFC-Flags
    SFCPause: BOOL;
    SFCReset: BOOL;
    
    // Indicadores de sincronizacion
    Ack: BOOL := TRUE;
    Execute: BOOL;
 
    // Entradas
    AlimentadorDelante: BOOL;
	PulsadorMarcha: BOOL; 
END_VAR
VAR_OUTPUT
    // Indicadores de sincronizacion
    Done: BOOL;
    Ready: BOOL;
	Fallo: BOOL;
    // Salidas
   AlimentadorAvanza: BOOL;
END_VAR
VAR
END_VAR

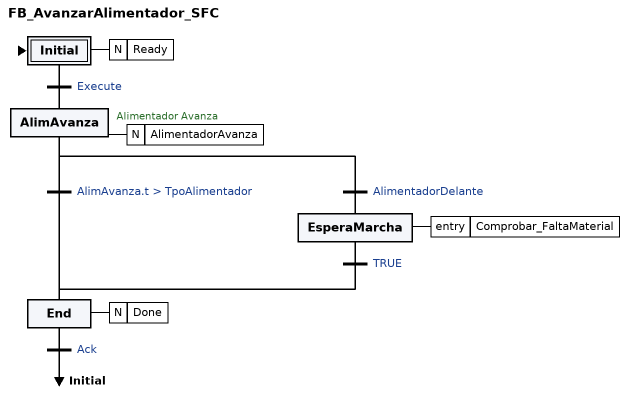
INITIAL_STEP Initial:
    Ready(N);
END_STEP
TRANSITION FROM Initial TO AlimAvanza
    := Execute;
END_TRANSITION
// Alimentador Avanza
STEP AlimAvanza:
    AlimentadorAvanza(N);
END_STEP
TRANSITION FROM AlimAvanza TO End
    := AlimAvanza.t > TpoAlimentador;
END_TRANSITION
TRANSITION FROM AlimAvanza TO EsperaMarcha
    := AlimentadorDelante;
END_TRANSITION
STEP EsperaMarcha:
    Comprobar_FaltaMaterial(P1);  // entry action
END_STEP
TRANSITION FROM EsperaMarcha TO End
    := TRUE;
END_TRANSITION
STEP End:
    Done(N);
END_STEP
TRANSITION FROM End TO Initial
    := Ack;
END_TRANSITION

ACTION Comprobar_FaltaMaterial:
FaltaMaterial := TRUE;
END_ACTION

END_FUNCTION_BLOCK

// ---- POUs/Tareas/FB_SituarPale_SFC.TcPOU
FUNCTION_BLOCK FB_SituarPale_SFC

VAR_IN_OUT
	  TpoPaleEntrada: TIME;
END_VAR

VAR_INPUT
    // SFC-Flags
    SFCPause: BOOL;
    SFCReset: BOOL;
    
    // Indicadores de sincronizacion
    Ack: BOOL := TRUE;
    Execute: BOOL;
    
    // Entradas
    PresenciaPale: BOOL;
    CodigoPaleBit0: BOOL;
    CodigoPaleBit1: BOOL;
    CodigoPaleBit2: BOOL;    
END_VAR
VAR_OUTPUT
    // Indicadores de sincronizacion
    Done: BOOL;
    Ready: BOOL;
    
    // Parametros
    CodigoPale: BYTE;
    
    // Salidas
    CintaActiva: BOOL;
END_VAR
VAR
END_VAR

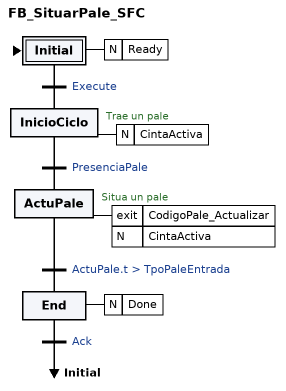
INITIAL_STEP Initial:
    Ready(N);
END_STEP
TRANSITION FROM Initial TO InicioCiclo
    := Execute;
END_TRANSITION
// Trae un pale
STEP InicioCiclo:
    CintaActiva(N);
END_STEP
TRANSITION FROM InicioCiclo TO ActuPale
    := PresenciaPale;
END_TRANSITION
// Situa un pale
STEP ActuPale:
    CodigoPale_Actualizar(P0);  // exit action
    CintaActiva(N);
END_STEP
TRANSITION FROM ActuPale TO End
    := ActuPale.t > TpoPaleEntrada;
END_TRANSITION
STEP End:
    Done(N);
END_STEP
TRANSITION FROM End TO Initial
    := Ack;
END_TRANSITION

ACTION CodigoPale_Actualizar:
CodigoPale.0 := CodigoPaleBit0;
CodigoPale.1 := CodigoPaleBit1;
CodigoPale.2 := CodigoPaleBit2;
END_ACTION

END_FUNCTION_BLOCK

// ---- POUs/Tareas/FB_CargarPieza_SFC.TcPOU
FUNCTION_BLOCK FB_CargarPieza_SFC

VAR_IN_OUT
	    TpoPinza: TIME;
END_VAR

VAR_INPUT
    // SFC-Flags
    SFCPause: BOOL;
    SFCReset: BOOL;
    
    // Indicadores de sincronizacion
    Ack: BOOL := TRUE;
    Execute: BOOL;
    
    // Entradas
    CargadorDetras : BOOL;
	CargadorDelante : BOOL;
	CargadorArriba : BOOL;
	CargadorAbajo : BOOL;  
END_VAR
VAR_OUTPUT
    // Indicadores de sincronizacion
    Done: BOOL;
    Ready: BOOL;
    
    // Salidas
    CargadorAvanza : BOOL;
	CargadorBaja : BOOL; 	
	CargadorCierra : BOOL;
END_VAR
VAR
END_VAR

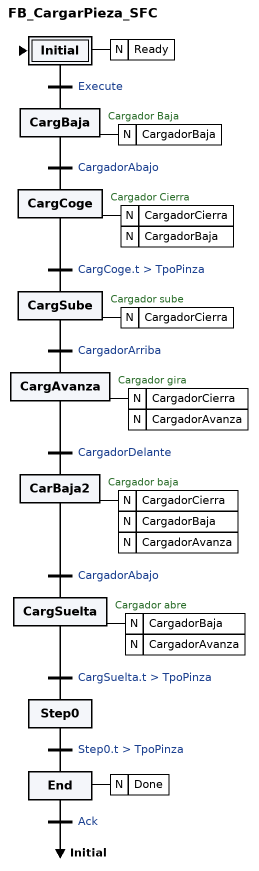
INITIAL_STEP Initial:
    Ready(N);
END_STEP
TRANSITION FROM Initial TO CargBaja
    := Execute;
END_TRANSITION
// Cargador Baja
STEP CargBaja:
    CargadorBaja(N);
END_STEP
TRANSITION FROM CargBaja TO CargCoge
    := CargadorAbajo;
END_TRANSITION
// Cargador Cierra
STEP CargCoge:
    CargadorCierra(N);
    CargadorBaja(N);
END_STEP
TRANSITION FROM CargCoge TO CargSube
    := CargCoge.t > TpoPinza;
END_TRANSITION
// Cargador sube
STEP CargSube:
    CargadorCierra(N);
END_STEP
TRANSITION FROM CargSube TO CargAvanza
    := CargadorArriba;
END_TRANSITION
// Cargador gira
STEP CargAvanza:
    CargadorCierra(N);
    CargadorAvanza(N);
END_STEP
TRANSITION FROM CargAvanza TO CarBaja2
    := CargadorDelante;
END_TRANSITION
// Cargador baja
STEP CarBaja2:
    CargadorCierra(N);
    CargadorBaja(N);
    CargadorAvanza(N);
END_STEP
TRANSITION FROM CarBaja2 TO CargSuelta
    := CargadorAbajo;
END_TRANSITION
// Cargador abre
STEP CargSuelta:
    CargadorBaja(N);
    CargadorAvanza(N);
END_STEP
TRANSITION FROM CargSuelta TO Step0
    := CargSuelta.t > TpoPinza;
END_TRANSITION
STEP Step0:
END_STEP
TRANSITION FROM Step0 TO End
    := Step0.t > TpoPinza;
END_TRANSITION
STEP End:
    Done(N);
END_STEP
TRANSITION FROM End TO Initial
    := Ack;
END_TRANSITION

END_FUNCTION_BLOCK

// ---- POUs/Tareas/FB_EmpujarPlato_SFC.TcPOU
FUNCTION_BLOCK FB_EmpujarPlato_SFC

VAR_IN_OUT
	   TpoEmpujadorAvanza: TIME;
END_VAR

VAR_INPUT
    // SFC-Flags
    SFCPause: BOOL;
    SFCReset: BOOL;
    
    // Indicadores de sincronizacion
    Ack: BOOL := TRUE;
    Execute: BOOL;
    
    
    // Entradas
   PlatoEmpujadorDetras : BOOL;
END_VAR
VAR_OUTPUT
    // Indicadores de sincronizacion
    Done: BOOL;
    Ready: BOOL;
    
    // Salidas
    PlatoEmpujadorAvanza : BOOL;
	PlatoRetenedorAtras : BOOL;
END_VAR
VAR
END_VAR

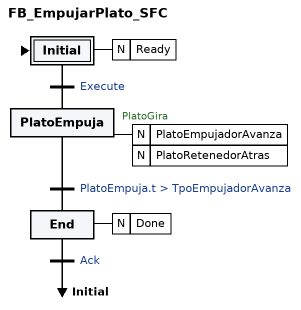
INITIAL_STEP Initial:
    Ready(N);
END_STEP
TRANSITION FROM Initial TO PlatoEmpuja
    := Execute;
END_TRANSITION
// PlatoGira
STEP PlatoEmpuja:
    PlatoEmpujadorAvanza(N);
    PlatoRetenedorAtras(N);
END_STEP
TRANSITION FROM PlatoEmpuja TO End
    := PlatoEmpuja.t > TpoEmpujadorAvanza;
END_TRANSITION
STEP End:
    Done(N);
END_STEP
TRANSITION FROM End TO Initial
    := Ack;
END_TRANSITION

END_FUNCTION_BLOCK

// ---- POUs/Tareas/FB_RetrocederPlato_SFC.TcPOU
FUNCTION_BLOCK FB_RetrocederPlato_SFC
VAR_IN_OUT
	   TpoEmpujadorAvanza: TIME;
END_VAR

VAR_INPUT
    // SFC-Flags
    SFCPause: BOOL;
    SFCReset: BOOL;
    
    // Indicadores de sincronizacion
    Ack: BOOL := TRUE;
    Execute: BOOL;
    
    // Entradas
   PlatoEmpujadorDetras : BOOL;
END_VAR
VAR_OUTPUT
    // Indicadores de sincronizacion
    Done: BOOL;
    Ready: BOOL;
    
    // Salidas
    PlatoEmpujadorAvanza : BOOL;
	PlatoRetenedorAtras : BOOL;
END_VAR
VAR
	S3: INT;
END_VAR

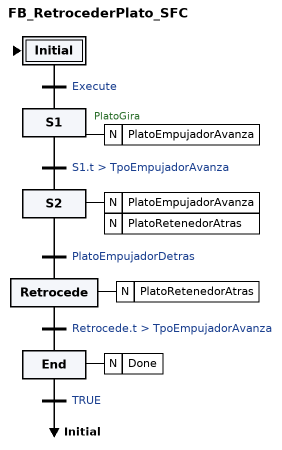
INITIAL_STEP Initial:
END_STEP
TRANSITION FROM Initial TO S1
    := Execute;
END_TRANSITION
// PlatoGira
STEP S1:
    PlatoEmpujadorAvanza(N);
END_STEP
TRANSITION FROM S1 TO S2
    := S1.t > TpoEmpujadorAvanza;
END_TRANSITION
STEP S2:
    PlatoEmpujadorAvanza(N);
    PlatoRetenedorAtras(N);
END_STEP
TRANSITION FROM S2 TO Retrocede
    := PlatoEmpujadorDetras;
END_TRANSITION
STEP Retrocede:
    PlatoRetenedorAtras(N);
END_STEP
TRANSITION FROM Retrocede TO End
    := Retrocede.t > TpoEmpujadorAvanza;
END_TRANSITION
STEP End:
    Done(N);
END_STEP
TRANSITION FROM End TO Initial
    := TRUE;
END_TRANSITION

END_FUNCTION_BLOCK

// ---- POUs/Tareas/FB_DescargarPieza_SFC.TcPOU
FUNCTION_BLOCK FB_DescargarPieza_SFC

VAR_IN_OUT
	    TpoPinza: TIME;
END_VAR

VAR_INPUT
    // SFC-Flags
    SFCPause: BOOL;
    SFCReset: BOOL;
    
    // Indicadores de sincronizacion
    Ack: BOOL := TRUE;
    Execute: BOOL;
    
    // Entradas
    DescargadorDetras : BOOL;
	DescargadorDelante : BOOL;
	DescargadorArriba : BOOL;
	DescargadorAbajo : BOOL;
END_VAR
VAR_OUTPUT
    // Indicadores de sincronizacion
    Done: BOOL;
    Ready: BOOL;
    
    // Salidas
    DescargadorAvanza AT %Q*: BOOL;
	DescargadorBaja AT %Q*: BOOL;
	DescargadorCierra AT %Q*: BOOL;
END_VAR
VAR
END_VAR

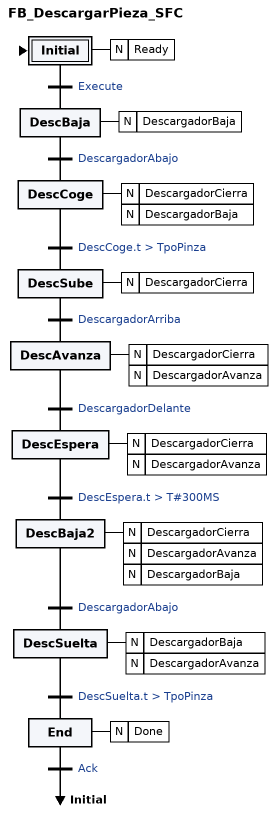
INITIAL_STEP Initial:
    Ready(N);
END_STEP
TRANSITION FROM Initial TO DescBaja
    := Execute;
END_TRANSITION
STEP DescBaja:
    DescargadorBaja(N);
END_STEP
TRANSITION FROM DescBaja TO DescCoge
    := DescargadorAbajo;
END_TRANSITION
STEP DescCoge:
    DescargadorCierra(N);
    DescargadorBaja(N);
END_STEP
TRANSITION FROM DescCoge TO DescSube
    := DescCoge.t > TpoPinza;
END_TRANSITION
STEP DescSube:
    DescargadorCierra(N);
END_STEP
TRANSITION FROM DescSube TO DescAvanza
    := DescargadorArriba;
END_TRANSITION
STEP DescAvanza:
    DescargadorCierra(N);
    DescargadorAvanza(N);
END_STEP
TRANSITION FROM DescAvanza TO DescEspera
    := DescargadorDelante;
END_TRANSITION
STEP DescEspera:
    DescargadorCierra(N);
    DescargadorAvanza(N);
END_STEP
TRANSITION FROM DescEspera TO DescBaja2
    := DescEspera.t > T#300MS;
END_TRANSITION
STEP DescBaja2:
    DescargadorCierra(N);
    DescargadorAvanza(N);
    DescargadorBaja(N);
END_STEP
TRANSITION FROM DescBaja2 TO DescSuelta
    := DescargadorAbajo;
END_TRANSITION
STEP DescSuelta:
    DescargadorBaja(N);
    DescargadorAvanza(N);
END_STEP
TRANSITION FROM DescSuelta TO End
    := DescSuelta.t > TpoPinza;
END_TRANSITION
STEP End:
    Done(N);
END_STEP
TRANSITION FROM End TO Initial
    := Ack;
END_TRANSITION

END_FUNCTION_BLOCK

// ---- POUs/Tareas/FB_RechazarPieza_SFC.TcPOU
FUNCTION_BLOCK FB_RechazarPieza_SFC

VAR_IN_OUT
	TpoRechazador: TIME;
END_VAR

VAR_INPUT
    // SFC-Flags
    SFCPause: BOOL;
    SFCReset: BOOL;
    
    // Indicadores de sincronizacion
    Ack: BOOL := TRUE;
    Execute: BOOL;
    
    // Entradas
    RechazadorDetras : BOOL;
	RechazadorDelante : BOOL;
	RechazadorArriba : BOOL;
	RechazadorVacio : BOOL;
	PulsadorMarcha: BOOL;
END_VAR
VAR_OUTPUT
    // Indicadores de sincronizacion
    Done: BOOL;
    Ready: BOOL;
	Fallo: BOOL;

    // Salidas
    RechazadorAvanza : BOOL;
	RechazadorRetrocede : BOOL;
	RechazadorBaja : BOOL;
	RechazadorSucciona : BOOL;
END_VAR
VAR
END_VAR

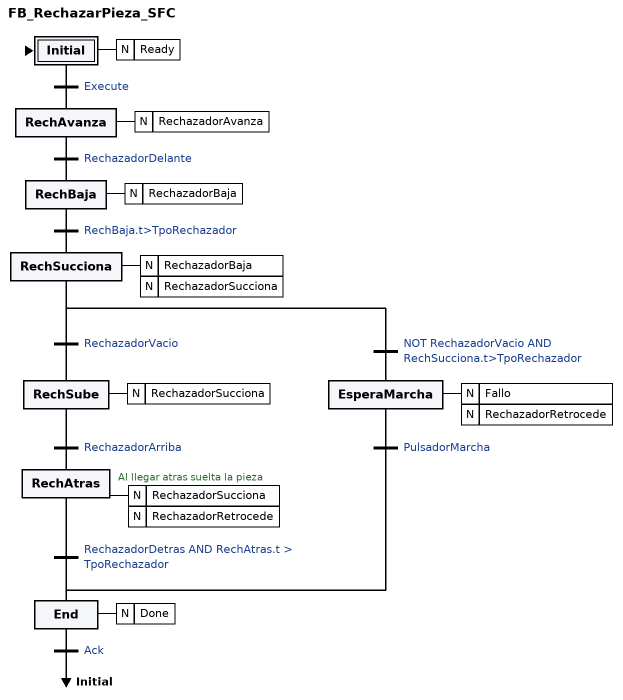
INITIAL_STEP Initial:
    Ready(N);
END_STEP
TRANSITION FROM Initial TO RechAvanza
    := Execute;
END_TRANSITION
STEP RechAvanza:
    RechazadorAvanza(N);
END_STEP
TRANSITION FROM RechAvanza TO RechBaja
    := RechazadorDelante;
END_TRANSITION
STEP RechBaja:
    RechazadorBaja(N);
END_STEP
TRANSITION FROM RechBaja TO RechSucciona
    := RechBaja.t>TpoRechazador;
END_TRANSITION
STEP RechSucciona:
    RechazadorBaja(N);
    RechazadorSucciona(N);
END_STEP
TRANSITION FROM RechSucciona TO RechSube
    := RechazadorVacio;
END_TRANSITION
STEP RechSube:
    RechazadorSucciona(N);
END_STEP
TRANSITION FROM RechSube TO RechAtras
    := RechazadorArriba;
END_TRANSITION
// Al llegar atras suelta la pieza
STEP RechAtras:
    RechazadorSucciona(N);
    RechazadorRetrocede(N);
END_STEP
TRANSITION FROM RechAtras TO End
    := RechazadorDetras AND RechAtras.t > TpoRechazador;
END_TRANSITION
TRANSITION FROM RechSucciona TO EsperaMarcha
    := NOT RechazadorVacio AND RechSucciona.t>TpoRechazador;
END_TRANSITION
STEP EsperaMarcha:
    Fallo(N);
    RechazadorRetrocede(N);
END_STEP
TRANSITION FROM EsperaMarcha TO End
    := PulsadorMarcha;
END_TRANSITION
STEP End:
    Done(N);
END_STEP
TRANSITION FROM End TO Initial
    := Ack;
END_TRANSITION

END_FUNCTION_BLOCK

// ---- POUs/Tareas/FB_TransferirPale_SFC.TcPOU
FUNCTION_BLOCK FB_TransferirPale_SFC

VAR_IN_OUT
	TpoCintaRetenedor: TIME;
    TpoPaleSalida: TIME;
    TpoPaleTransferencia: TIME;
END_VAR


VAR_INPUT
    // SFC-Flags
    SFCPause: BOOL;
    SFCReset: BOOL;
    
    // Indicadores de sincronizacion
    Ack: BOOL := TRUE;
    Execute: BOOL;
    
    // Entradas
    PresenciaPale: BOOL;
END_VAR
VAR_OUTPUT
    // Indicadores de sincronizacion
    Done: BOOL;
    Ready: BOOL;
    // Salidas
    CintaActiva: BOOL;
    RetenedorBaja: BOOL;
	SeparadorSube: BOOL;
END_VAR
VAR
END_VAR

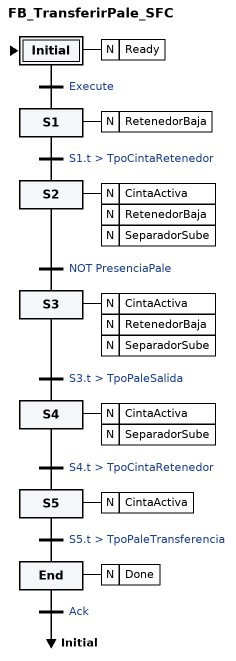
INITIAL_STEP Initial:
    Ready(N);
END_STEP
TRANSITION FROM Initial TO S1
    := Execute;
END_TRANSITION
STEP S1:
    RetenedorBaja(N);
END_STEP
TRANSITION FROM S1 TO S2
    := S1.t > TpoCintaRetenedor;
END_TRANSITION
STEP S2:
    CintaActiva(N);
    RetenedorBaja(N);
    SeparadorSube(N);
END_STEP
TRANSITION FROM S2 TO S3
    := NOT PresenciaPale;
END_TRANSITION
STEP S3:
    CintaActiva(N);
    RetenedorBaja(N);
    SeparadorSube(N);
END_STEP
TRANSITION FROM S3 TO S4
    := S3.t > TpoPaleSalida;
END_TRANSITION
STEP S4:
    CintaActiva(N);
    SeparadorSube(N);
END_STEP
TRANSITION FROM S4 TO S5
    := S4.t > TpoCintaRetenedor;
END_TRANSITION
STEP S5:
    CintaActiva(N);
END_STEP
TRANSITION FROM S5 TO End
    := S5.t > TpoPaleTransferencia;
END_TRANSITION
STEP End:
    Done(N);
END_STEP
TRANSITION FROM End TO Initial
    := Ack;
END_TRANSITION

END_FUNCTION_BLOCK

// ---- POUs/Tareas/FB_Medir_SFC.TcPOU
FUNCTION_BLOCK FB_Medir_SFC
VAR_IN_OUT
    ListadePiezas : ARRAY[1..TAMANO_LISTA_PIEZAS] OF Pieza; 
	TpoMedidor: TIME;
    
END_VAR
VAR_INPUT
    // SFC-Flags
    SFCPause: BOOL;
    SFCReset: BOOL;
    
    // Indicadores de sincronizacion
    Ack: BOOL := TRUE;
    Execute: BOOL;
    
    // Parametros
	NCiclos: INT ;
	AUX_Medidor: INT;
	AUX_FotoElectrico: INT;
	AUX_Metalico: INT;
	
    
    // Entradas
    DetectorInductivo: BOOL;
	DetectorFotoelectrico: BOOL;
	Codificador: UINT;
END_VAR
VAR_OUTPUT
    // Indicadores de sincronizacion
    Done: BOOL;
    Ready: BOOL;
    
    // Salidas
   MedidorBaja: BOOL;
END_VAR
VAR
END_VAR

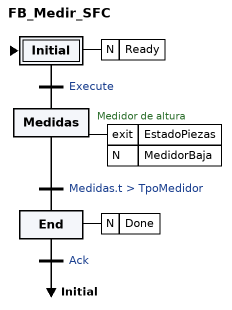
INITIAL_STEP Initial:
    Ready(N);
END_STEP
TRANSITION FROM Initial TO Medidas
    := Execute;
END_TRANSITION
// Medidor de altura
STEP Medidas:
    EstadoPiezas(P0);  // exit action
    MedidorBaja(N);
END_STEP
TRANSITION FROM Medidas TO End
    := Medidas.t > TpoMedidor;
END_TRANSITION
STEP End:
    Done(N);
END_STEP
TRANSITION FROM End TO Initial
    := Ack;
END_TRANSITION

ACTION EstadoPiezas:

//Medidor de altura
AUX_Medidor := AjustarIndice(Nciclos) ;
ListadePiezas[AUX_Medidor].BienColocada := Codificador < 1600; 
ListadePiezas[AUX_Medidor].TipoPieza.Alta := Codificador < 1310;

//Fotoelectrioco
AUX_FotoElectrico := AjustarIndice(Nciclos - 1);
ListadePiezas[AUX_FotoElectrico].TipoPieza.Claro := DetectorFotoelectrico; //TRUE si es clara


//Inductivo
AUX_Metalico := AjustarIndice(Nciclos - 2);
ListadePiezas[AUX_Metalico].TipoPieza.Metalico :=  DetectorInductivo; //TRUE si metalica
END_ACTION

END_FUNCTION_BLOCK

// ---- GlobalTextList.TcGTLO
TEXTLIST GlobalTextList
  918 = '%d'
  602 = '%s'
  1040 = '+'
  1168 = '-'
  100 = '.0'
  767 = '.1'
  53 = '.2'
  247 = '.3'
  425 = '0'
  454 = '1'
  355 = '2'
  317 = '3'
  39 = '4'
  859 = '<'
  973 = '>'
  729 = 'A Ciclos'
  145 = 'A Piezas'
  515 = 'A+'
  281 = 'A-'
  359 = 'ACiclos'
  568 = 'Alar'
  350 = 'Alarma'
  301 = 'ALARMA'
  30 = 'Ali delante'
  32 = 'Alim. Avanza'
  328 = 'Alimen Avanz'
  136 = 'Alimentador'
  956 = 'ALIMENTADOR DE TAPAS'
  364 = 'Alta'
  363 = 'alta'
  743 = 'Alto'
  639 = 'Altura'
  34 = 'B+'
  831 = 'Baja'
  984 = 'Bajo'
  590 = 'Blanca'
  452 = 'BLANCA'
  354 = 'C+'
  1133 = 'Cargador'
  228 = 'CI'
  318 = 'Ciclo'
  144 = 'Ciclo a Ciclo'
  1109 = 'Ciclo-Ciclo'
  150 = 'CicloACiclo'
  1218 = 'Cinta'
  1471 = 'Clara'
  528 = 'CM'
  46 = 'CN'
  737 = 'Comenzar'
  875 = 'Conect'
  143 = 'Conectada'
  409 = 'conectada'
  216 = 'cp'
  24 = 'CR'
  897 = 'CV'
  159 = 'D+'
  358 = 'D.F.'
  412 = 'D.I.'
  87 = 'Desconect'
  416 = 'Desconectada'
  366 = 'Desechar'
  742 = 'df'
  545 = 'di'
  420 = 'DPO'
  90 = 'E+'
  910 = 'E-Stop'
  820 = 'E-Stp'
  503 = 'Emerg'
  942 = 'EMERGENCIA'
  813 = 'Emp. Plato'
  1157 = 'Empujador'
  862 = 'Entrada Palé'
  1274 = 'Eyector'
  127 = 'F+'
  1439 = 'F-'
  668 = 'Finalizar'
  1290 = 'FinCiclo'
  353 = 'FM'
  1156 = 'FMS-205: ALIMENTADOR DE TAPAS'
  1085 = 'G+'
  352 = 'H+'
  1031 = 'Hidrúlico'
  437 = 'Hor. Carga'
  265 = 'Hor. Descarg.'
  620 = 'Hor. Rechazo'
  1456 = 'I+'
  636 = 'J+'
  1293 = 'K+'
  726 = 'K-'
  184 = 'L+'
  628 = 'lamparamarcha'
  583 = 'Limpiar'
  177 = 'LimpiarTapas'
  635 = 'luz alarma'
  323 = 'luzmarcha'
  289 = 'MAN'
  937 = 'Manual ON'
  163 = 'Marcha'
  357 = 'Material'
  356 = 'Medidor'
  547 = 'METAL'
  965 = 'Metálica'
  1068 = 'MODO'
  101 = 'Negra'
  325 = 'NEGRA'
  838 = 'pale'
  943 = 'Pale'
  199 = 'Panel'
  561 = 'Parada'
  584 = 'PARÁMETROS'
  241 = 'Pausa'
  936 = 'Pendientes'
  766 = 'Pinza'
  29 = 'Pinza Carga'
  1127 = 'Pinza Descarg.'
  129 = 'Planta'
  1057 = 'PLANTA'
  4 = 'POC'
  85 = 'pp'
  74 = 'ppp'
  1135 = 'Preparar'
  258 = 'Protector'
  493 = 'PV'
  759 = 'R+'
  892 = 'R-'
  732 = 'Realizadas'
  1099 = 'Rechazar'
  821 = 'Reset'
  796 = 'Reten. plato'
  190 = 'Retenedor'
  656 = 'REV'
  343 = 'RUN'
  800 = 'S+'
  529 = 'S-'
  949 = 'Salida Palé'
  277 = 'Selec Man'
  1155 = 'Sensores'
  538 = 'Solicitadas'
  879 = 'sonoro'
  990 = 'Sonoro'
  827 = 'Succiona'
  1236 = 'Tarea'
  390 = 'TAREA'
  1506 = 'Tipo'
  198 = 'TIPO'
  569 = 'Transf. Palé'
  1294 = 'V+'
  368 = 'Vaciar'
  178 = 'Ver. Carga'
  725 = 'Ver. Descarg.'
  153 = 'Ver. Rechazo'
END_TEXTLIST

// ---- VISUs/Visualization.TcVIS
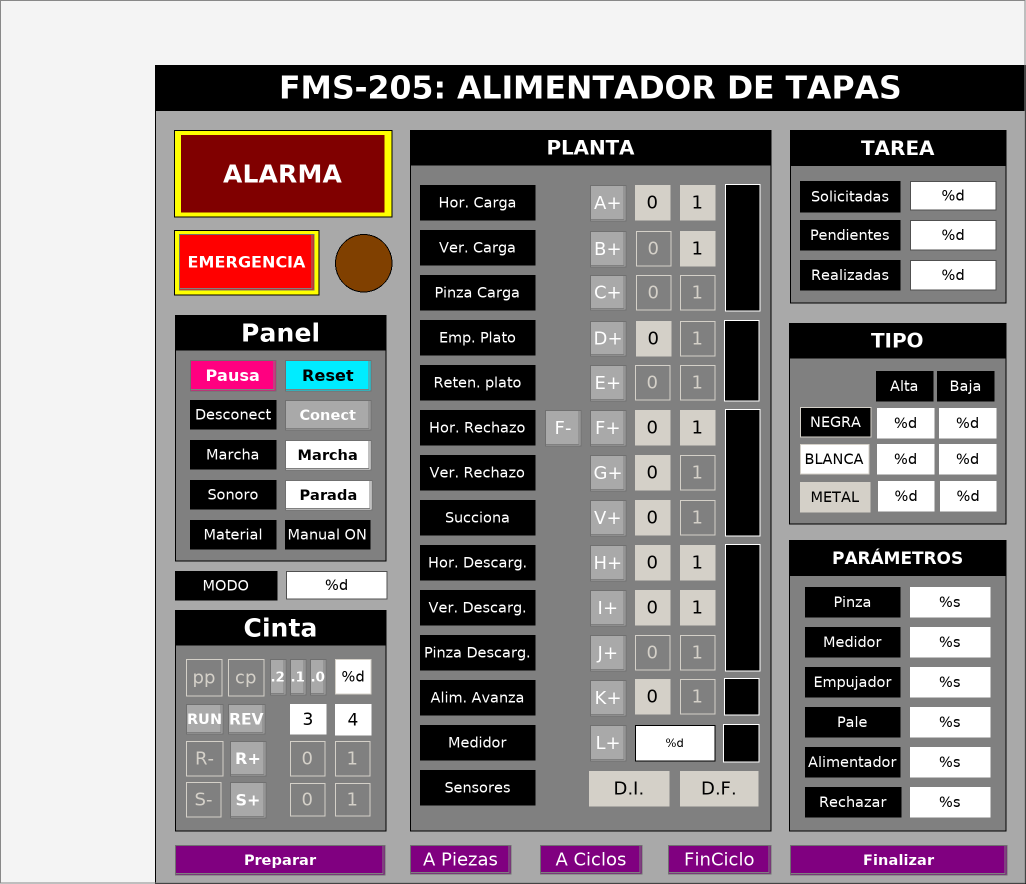
VISUALIZATION Visualization  // 1026x884
    Rectangle (155,110 871x774)
    Rectangle (175,315 211x246)
    Rectangle (410,160 361x671)
    Rectangle (420,185 115x35), "Hor. Carga"
    Rectangle (420,230 115x35), "Ver. Carga"
        toggle MAIN.Estacion.CargadorCierra
    Rectangle (420,275 115x35), "Pinza Carga"
    Rectangle (420,320 115x35), "Emp. Plato"
    Rectangle (420,365 115x35), "Reten. plato"
    Rectangle (420,410 115x35), "Hor. Rechazo"
    Rectangle (420,680 115x35), "Alim. Avanza"
    Rectangle (420,455 115x35), "Ver. Rechazo"
    Rectangle (420,500 115x35), "Succiona"
    Rectangle (420,545 115x35), "Hor. Descarg."
    Rectangle (420,590 115x35), "Ver. Descarg."
    Rectangle (420,635 115x35), "Pinza Descarg."
    Rectangle (420,725 115x35), "Medidor"
    Button (590,185 36x36), "A+", colour toggle: MAIN.Estacion.CargadorAvanza
        toggle MAIN.Estacion.CargadorAvanza
    Button (590,231 36x36), "B+", colour toggle: MAIN.Estacion.CargadorBaja
        toggle MAIN.Estacion.CargadorBaja
    Button (590,275 36x35), "C+", colour toggle: MAIN.Estacion.CargadorCierra
        toggle MAIN.Estacion.CargadorCierra
    Button (590,321 36x35), "D+", colour toggle: MAIN.Estacion.PlatoEmpujadorAvanza
        toggle MAIN.Estacion.PlatoEmpujadorAvanza
    Button (590,545 36x36), "H+", colour toggle: MAIN.Estacion.DescargadorAvanza
        toggle MAIN.Estacion.DescargadorAvanza
    Button (590,365 36x36), "E+", colour toggle: MAIN.Estacion.PlatoRetenedorAtras
        toggle MAIN.Estacion.PlatoRetenedorAtras
    Button (590,410 36x36), "F+", colour toggle: MAIN.Estacion.RechazadorAvanza
        toggle MAIN.Estacion.RechazadorAvanza
    Button (590,455 36x36), "G+", colour toggle: MAIN.Estacion.RechazadorBaja
        toggle MAIN.Estacion.RechazadorBaja
    Button (545,410 36x36), "F-", colour toggle: MAIN.Estacion.RechazadorRetrocede
        toggle MAIN.Estacion.RechazadorRetrocede
    Button (590,590 36x36), "I+", colour toggle: MAIN.Estacion.DescargadorAbajo
        toggle MAIN.Estacion.DescargadorAbajo
    Button (590,500 36x36), "V+", colour toggle: MAIN.Estacion.RechazadorSucciona
        toggle MAIN.Estacion.RechazadorSucciona
    Button (590,635 36x36), "J+", colour toggle: MAIN.Estacion.DescargadorCierra
        toggle MAIN.Estacion.DescargadorCierra
    Button (590,725 36x36), "L+", colour toggle: MAIN.Estacion.MedidorBaja
        toggle MAIN.Estacion.MedidorBaja
    Rectangle (410,130 361x35), "PLANTA"
    Button (285,440 86x30), "Marcha", colour toggle: MAIN.Estacion.PulsadorMarcha
        tap MAIN.Estacion.PulsadorMarcha
        toggle MAIN.Estacion.PulsadorMarcha
    Button (285,400 86x30), "Conect", colour toggle: MAIN.Estacion.EstacionConectada
        toggle MAIN.Estacion.EstacionConectada
    Rectangle (175,315 211x35), "Panel"
    Rectangle (789,323 217x201)
    Rectangle (789,323 217x35), "TIPO"
    Rectangle (175,620 211x211)
    Button (186,704 37x30), "RUN", colour toggle: MAIN.Estacion.CintaActiva
        toggle MAIN.Estacion.CintaActiva
    Button (228,704 37x30), "REV", colour toggle: MAIN.Estacion.CintaInvierte
        toggle MAIN.Estacion.CintaInvierte
    Rectangle (175,610 211x35), "Cinta"
    Rectangle (420,770 115x35), "Sensores"
    Rectangle (155,65 871x45), "FMS-205: ALIMENTADOR DE TAPAS"
    Rectangle (635,185 35x35), "0", colour toggle: MAIN.Estacion.CargadorDetras
    Rectangle (680,185 35x35), "1", colour toggle: MAIN.Estacion.CargadorDelante
    Rectangle (725,184 35x127), colour toggle: MAIN.Estacion.CargarPieza.Execute
    Rectangle (636,231 35x35), "0", colour toggle: MAIN.Estacion.CargadorAbajo
    Rectangle (680,231 35x35), "1", colour toggle: MAIN.Estacion.CargadorArriba
    Rectangle (636,275 35x35), "0"
    Rectangle (680,275 35x35), "1"
    Rectangle (635,410 35x35), "0", colour toggle: MAIN.Estacion.RechazadorDetras
    Rectangle (636,321 35x35), "0", colour toggle: MAIN.Estacion.PlatoEmpujadorDetras
    Rectangle (680,321 35x35), "1"
    Rectangle (724,320 35x81), colour toggle: MAIN.Estacion.EmpujarPlato.Execute
    Rectangle (635,365 35x35), "0"
    Rectangle (680,365 35x35), "1"
    Rectangle (680,410 35x35), "1", colour toggle: MAIN.Estacion.RechazadorDelante
    Rectangle (725,409 35x127), colour toggle: MAIN.Estacion.RechazarPieza.Execute
    Rectangle (635,545 35x35), "0", colour toggle: MAIN.Estacion.DescargadorDetras
    Rectangle (635,455 35x35), "0", colour toggle: MAIN.Estacion.RechazadorArriba
    Rectangle (680,455 35x35), "1"
    Rectangle (635,500 35x35), "0", colour toggle: MAIN.Estacion.RechazadorVacio
    Rectangle (680,500 35x35), "1"
    Rectangle (680,545 35x35), "1", colour toggle: MAIN.Estacion.DescargadorDelante
    Rectangle (725,544 35x127), colour toggle: MAIN.Estacion.DescargarPieza.Execute
    Rectangle (635,679 35x35), "0", colour toggle: MAIN.Estacion.AlimentadorDelante
    Rectangle (635,590 35x35), "0", colour toggle: MAIN.Estacion.DescargadorAbajo
    Rectangle (680,590 35x35), "1", colour toggle: MAIN.Estacion.DescargadorArriba
    Rectangle (635,635 35x35), "0"
    Rectangle (680,635 35x35), "1"
    Rectangle (680,679 35x35), "1"
    Rectangle (724,678 35x37), colour toggle: MAIN.Estacion.AvanzarAlimentador.Execute
    Rectangle (723,724 36x38), colour toggle: MAIN.Estacion.Medir.Execute
    Button (230,741 36x35), "R+", colour toggle: MAIN.Estacion.RetenedorBaja
        toggle MAIN.Estacion.RetenedorBaja
    Button (230,782 36x36), "S+"
        toggle MAIN.Estacion.SeparadorSube
    Button (270,659 16x36), ".2", colour toggle: MAIN.Estacion.CodigoPaleBit2
        toggle MAIN.Estacion.CodigoPaleBit2
    Button (290,659 16x36), ".1", colour toggle: MAIN.Estacion.CodigoPaleBit1
        toggle MAIN.Estacion.CodigoPaleBit1
    Button (310,659 16x36), ".0", colour toggle: MAIN.Estacion.CodigoPaleBit0
        toggle MAIN.Estacion.CodigoPaleBit0
    Rectangle (290,741 35x35), "0"
    Rectangle (335,741 35x35), "1"
    Rectangle (290,783 35x33), "0"
    Rectangle (335,783 35x33), "1"
    Rectangle (186,741 37x35), "R-"
    Rectangle (186,782 35x35), "S-"
    Rectangle (285,520 85x29), "Manual ON", colour toggle: MAIN.Estacion.SelectorManual
    Button (285,480 87x30), "Parada", colour toggle: MAIN.Estacion.PulsadorParada
        toggle MAIN.Estacion.PulsadorParada
    Rectangle (190,520 86x29), "Material", colour toggle: MAIN.Estacion.LamparaMaterial
    Button (590,680 36x36), "K+", colour toggle: MAIN.Estacion.AlimentadorAvanza
        toggle MAIN.Estacion.AlimentadorAvanza
    Rectangle (635,725 80x36), "%d", text variable: MAIN.Estacion.Codificador
    Rectangle (290,704 36x30), "3", colour toggle: MAIN.Estacion.CintaActiva AND MAIN.Estacion.CintaInvierte
    Rectangle (335,704 36x31), "4", colour toggle: MAIN.Estacion.CintaActiva AND NOT MAIN.Estacion.CintaInvierte
    Rectangle (789,540 217x36), "PARÁMETROS"
    Rectangle (789,575 217x256)
    RoundedRectangle (805,667 95x30), "Empujador"
    RoundedRectangle (805,707 95x30), "Pale"
    RoundedRectangle (805,747 95x30), "Alimentador"
    RoundedRectangle (805,787 96x30), "Rechazar"
    Rectangle (910,667 80x30), "%s", text variable: MAIN.Estacion.TpoEmpujadorAvanza
        OnMouseClick: write the text variable via Default
    Rectangle (910,707 80x30), "%s", text variable: MAIN.Estacion.TpoPaleEntrada
        OnMouseClick: write the text variable via Default
    Rectangle (910,747 80x30), "%s", text variable: MAIN.Estacion.TpoAlimentador
        OnMouseClick: write the text variable via Default
    Rectangle (910,787 80x30), "%s", text variable: MAIN.Estacion.TpoRechazador
        OnMouseClick: write the text variable via Default
    RoundedRectangle (805,627 95x30), "Medidor"
    RoundedRectangle (805,587 95x30), "Pinza"
    Rectangle (910,587 80x30), "%s", text variable: MAIN.Estacion.TpoPinza
        OnMouseClick: write the text variable via Default
    Rectangle (910,627 80x30), "%s", text variable: MAIN.Estacion.TpoMedidor
        OnMouseClick: write the text variable via Default
    Rectangle (790,130 216x36), "TAREA"
    Rectangle (790,165 216x138)
    RoundedRectangle (800,181 100x31), "Solicitadas"
    Rectangle (910,181 86x29), "%d", text variable: MAIN.Estacion.UnidadesSolicitadas
        OnMouseClick: write the text variable via Default
    RoundedRectangle (800,220 100x30), "Pendientes"
    Rectangle (910,220 86x30), "%d", text variable: MAIN.Estacion.UnidadesPendientes
        OnMouseClick: write the text variable via Default
    RoundedRectangle (800,260 100x30), "Realizadas"
    Rectangle (910,260 86x30), "%d", text variable: MAIN.Estacion.UnidadesRealizadas
        OnMouseClick: write the text variable via Default
    Rectangle (877,408 57x30), "%d", text variable: MAIN.Estacion.ListaPiezasSolicitadas[1]
        OnMouseClick: write the text variable via Default
    Rectangle (877,444 57x30), "%d", text variable: MAIN.Estacion.ListaPiezasSolicitadas[2]
        OnMouseClick: write the text variable via Default
    Rectangle (878,481 56x30), "%d", text variable: MAIN.Estacion.ListaPiezasSolicitadas[3]
        OnMouseClick: write the text variable via Default
    Button (540,845 102x29), "A Ciclos", colour toggle: MAIN.Estacion.CicloACiclo
        toggle MAIN.Estacion.CicloACiclo
    Button (190,360 86x31), "Pausa", colour toggle: MAIN.Estacion.PausaEstado
        toggle MAIN.Estacion.PausaEstado
    Button (285,360 86x31), "Reset", colour toggle: MAIN.Estacion.ReiniciaEstado
        tap MAIN.Estacion.ReiniciaEstado
    Rectangle (335,659 36x35), "%d", text variable: MAIN.Estacion.CodigoPale
    Rectangle (589,771 80x35), "D.I.", colour toggle: MAIN.Estacion.DetectorInductivo
    Rectangle (680,771 78x35), "D.F.", colour toggle: MAIN.Estacion.DetectorFotoelectrico
    RoundedRectangle (800,407 71x30), "NEGRA"
    RoundedRectangle (800,444 69x30), "BLANCA"
    RoundedRectangle (800,482 70x30), "METAL"
    RoundedRectangle (876,371 57x30), "Alta"
    RoundedRectangle (937,371 57x30), "Baja"
    Rectangle (939,408 57x30), "%d", text variable: MAIN.Estacion.ListaPiezasSolicitadas[4]
        OnMouseClick: write the text variable via Default
    Rectangle (939,444 57x30), "%d", text variable: MAIN.Estacion.ListaPiezasSolicitadas[5]
        OnMouseClick: write the text variable via Default
    Rectangle (940,481 56x30), "%d", text variable: MAIN.Estacion.ListaPiezasSolicitadas[6]
        OnMouseClick: write the text variable via Default
    Rectangle (186,659 36x37), "pp", text variable: MAIN.Estacion.PresenciaPale
    Rectangle (228,659 36x37), "cp"
    Rectangle (190,440 86x29), "Marcha", colour toggle: MAIN.Estacion.LamparaMarcha
    Rectangle (190,400 86x29), "Desconect", colour toggle: MAIN.Estacion.DesconectaEstacion
    Rectangle (190,480 86x29), "Sonoro", colour toggle: MAIN.Estacion.AvisadorSonoro
    Rectangle (174,130 218x87)
    Rectangle (180,134 205x79), "ALARMA", colour toggle: MAIN.Estacion.LamparaAlarma
    Rectangle (174,230 145x65)
    Button (179,234 135x56), "EMERGENCIA", colour toggle: MAIN.Estacion.PulsadorEmergencia
        toggle MAIN.Estacion.PulsadorEmergencia
    Rectangle (286,571 101x28), "%d", text variable: MAIN.Estacion.Director.Modo
        OnMouseClick: write the text variable via Default
    Rectangle (175,571 102x29), "MODO"
    Button (668,845 103x29), "FinCiclo", colour toggle: MAIN.Estacion.FinCiclo
        toggle MAIN.Estacion.FinCiclo
    Button (175,845 210x30), "Preparar", colour toggle: MAIN.Estacion.PrepararProduccion
        toggle MAIN.Estacion.PrepararProduccion
    Button (790,845 217x30), "Finalizar", colour toggle: MAIN.Estacion.FinalizarProduccion
        toggle MAIN.Estacion.FinalizarProduccion
    Ellipse (335,234 57x58), colour toggle: MAIN.Estacion.Director.Defecto
    Button (410,845 101x29), "A Piezas", colour toggle: MAIN.Estacion.PiezaAPieza
        toggle MAIN.Estacion.PiezaAPieza
END_VISUALIZATION
